LIN {X 0,Y 467.53,Z 286.872,A -85,B 0,C 180,E1 -7582.074,E2 -7582.074} C_VEL
LIN {X 0,Y 467.591,Z 286.865,A -85,B 0,C 180,E1 -7584.888,E2 -7584.888} C_VEL
LIN {X 0,Y 467.615,Z 286.865,A -85,B 0,C 180,E1 -7587.769,E2 -7587.769} C_VEL
LIN {X 0,Y 467.564,Z 286.872,A -85,B 0,C 180,E1 -7591.045,E2 -7591.045} C_VEL
LIN {X 0,Y 467.584,Z 286.87,A -85,B 0,C 180,E1 -7594.242,E2 -7594.242} C_VEL
LIN {X 0,Y 467.545,Z 286.875,A -85,B 0,C 180,E1 -7597.186,E2 -7597.186} C_VEL
LIN {X 0,Y 467.569,Z 286.869,A -85,B 0,C 180,E1 -7600.265,E2 -7600.265} C_VEL
LIN {X 0,Y 467.548,Z 286.875,A -85,B 0,C 180,E1 -7603.745,E2 -7603.745} C_VEL
LIN {X 0,Y 467.586,Z 286.882,A -85,B 0,C 180,E1 -7605.055,E2 -7605.055} C_VEL
LIN {X 0,Y 468.088,Z 290.387,A -85,B 0,C 180,E1 -7607.496,E2 -7607.496} C_VEL
LIN {X 0,Y 468.175,Z 293.918,A -85,B 0,C 180,E1 -7609.798,E2 -7609.798} C_VEL
LIN {X 0,Y 467.977,Z 298.652,A -85,B 0,C 180,E1 -7612.744,E2 -7612.744} C_VEL
LIN {X 0,Y 467.777,Z 303.629,A -85,B 0,C 180,E1 -7615.724,E2 -7615.724} C_VEL
LIN {X 0,Y 467.533,Z 309.782,A -85,B 0,C 180,E1 -7619.264,E2 -7619.264} C_VEL
LIN {X 0,Y 467.277,Z 315.091,A -85,B 0,C 180,E1 -7622.209,E2 -7622.209} C_VEL
LIN {X 0,Y 467.138,Z 320.41,A -85,B 0,C 180,E1 -7625.086,E2 -7625.086} C_VEL
LIN {X 0,Y 466.974,Z 326.319,A -85,B 0,C 180,E1 -7628.206,E2 -7628.206} C_VEL
LIN {X 0,Y 471.454,Z 343.046,A -85,B 0,C 180,E1 -7628.788,E2 -7628.788} C_VEL
LIN {X 0,Y 473.649,Z 353.438,A -85,B 0,C 180,E1 -7629.228,E2 -7629.228} C_VEL
LIN {X 0,Y 473.146,Z 366.892,A -85,B 0,C 180,E1 -7629.767,E2 -7629.767} C_VEL
LIN {X 0,Y 472.348,Z 380.121,A -85,B 0,C 180,E1 -7630.441,E2 -7630.441} C_VEL
LIN {X 0,Y 471.548,Z 393.604,A -85,B 0,C 180,E1 -7631.311,E2 -7631.311} C_VEL
LIN {X 0,Y 470.665,Z 407.326,A -85,B 0,C 180,E1 -7632.4,E2 -7632.4} C_VEL
LIN {X 0,Y 469.85,Z 419.744,A -85,B 0,C 180,E1 -7633.601,E2 -7633.601} C_VEL
LIN {X 0,Y 469.066,Z 430.152,A -85,B 0,C 180,E1 -7634.799,E2 -7634.799} C_VEL
LIN {X 0,Y 468.451,Z 439.813,A -85,B 0,C 180,E1 -7636.111,E2 -7636.111} C_VEL
LIN {X 0,Y 467.819,Z 448.806,A -85,B 0,C 180,E1 -7637.55,E2 -7637.55} C_VEL
LIN {X 0,Y 467.464,Z 457.202,A -85,B 0,C 180,E1 -7639.168,E2 -7639.168} C_VEL
LIN {X 0,Y 467.052,Z 464.577,A -85,B 0,C 180,E1 -7640.909,E2 -7640.909} C_VEL
LIN {X 0,Y 466.824,Z 470.426,A -85,B 0,C 180,E1 -7642.648,E2 -7642.648} C_VEL
LIN {X 0,Y 466.726,Z 473.902,A -85,B 0,C 180,E1 -7643.949,E2 -7643.949} C_VEL
LIN {X 0,Y 466.617,Z 477.414,A -85,B 0,C 180,E1 -7645.681,E2 -7645.681} C_VEL
LIN {X 0,Y 466.638,Z 479.725,A -85,B 0,C 180,E1 -7647.41,E2 -7647.41} C_VEL
LIN {X 0,Y 466.586,Z 480.888,A -85,B 0,C 180,E1 -7649.137,E2 -7649.137} C_VEL
LIN {X 0,Y 466.586,Z 480.887,A -85,B 0,C 180,E1 -7650.863,E2 -7650.863} C_VEL
LIN {X 0,Y 466.638,Z 479.722,A -85,B 0,C 180,E1 -7652.589,E2 -7652.589} C_VEL
LIN {X 0,Y 466.617,Z 477.411,A -85,B 0,C 180,E1 -7654.319,E2 -7654.319} C_VEL
LIN {X 0,Y 466.751,Z 473.905,A -85,B 0,C 180,E1 -7656.05,E2 -7656.05} C_VEL
LIN {X 0,Y 466.862,Z 469.113,A -85,B 0,C 180,E1 -7657.786,E2 -7657.786} C_VEL
LIN {X 0,Y 467.115,Z 462.905,A -85,B 0,C 180,E1 -7659.526,E2 -7659.526} C_VEL
LIN {X 0,Y 467.59,Z 455.107,A -85,B 0,C 180,E1 -7661.267,E2 -7661.267} C_VEL
LIN {X 0,Y 467.983,Z 446.593,A -85,B 0,C 180,E1 -7662.833,E2 -7662.833} C_VEL
LIN {X 0,Y 468.659,Z 436.814,A -85,B 0,C 180,E1 -7664.325,E2 -7664.325} C_VEL
LIN {X 0,Y 469.317,Z 426.585,A -85,B 0,C 180,E1 -7665.637,E2 -7665.637} C_VEL
LIN {X 0,Y 470.163,Z 414.572,A -85,B 0,C 180,E1 -7666.928,E2 -7666.928} C_VEL
LIN {X 0,Y 470.985,Z 402.163,A -85,B 0,C 180,E1 -7668.036,E2 -7668.036} C_VEL
LIN {X 0,Y 471.84,Z 388.848,A -85,B 0,C 180,E1 -7669.015,E2 -7669.015} C_VEL
LIN {X 0,Y 472.717,Z 374.15,A -85,B 0,C 180,E1 -7669.882,E2 -7669.882} C_VEL
LIN {X 0,Y 473.379,Z 360.05,A -85,B 0,C 180,E1 -7670.527,E2 -7670.527} C_VEL
LIN {X 0,Y 473.507,Z 352.11,A -85,B 0,C 180,E1 -7670.827,E2 -7670.827} C_VEL
LIN {X 0,Y 469.977,Z 337.263,A -85,B 0,C 180,E1 -7671.427,E2 -7671.427} C_VEL
LIN {X 0,Y 466.957,Z 326.298,A -85,B 0,C 180,E1 -7671.815,E2 -7671.815} C_VEL
LIN {X 0,Y 467.136,Z 320.455,A -85,B 0,C 180,E1 -7674.913,E2 -7674.913} C_VEL
LIN {X 0,Y 467.277,Z 315.165,A -85,B 0,C 180,E1 -7677.79,E2 -7677.79} C_VEL
LIN {X 0,Y 467.536,Z 309.843,A -85,B 0,C 180,E1 -7680.735,E2 -7680.735} C_VEL
LIN {X 0,Y 467.774,Z 303.655,A -85,B 0,C 180,E1 -7684.276,E2 -7684.276} C_VEL
LIN {X 0,Y 467.974,Z 298.65,A -85,B 0,C 180,E1 -7687.255,E2 -7687.255} C_VEL
LIN {X 0,Y 468.172,Z 293.896,A -85,B 0,C 180,E1 -7690.202,E2 -7690.202} C_VEL
LIN {X 0,Y 468.082,Z 290.182,A -85,B 0,C 180,E1 -7692.633,E2 -7692.633} C_VEL
LIN {X 0,Y 467.585,Z 286.869,A -85,B 0,C 180,E1 -7695.055,E2 -7695.055} C_VEL
LIN {X 0,Y 467.583,Z 286.87,A -85,B 0,C 180,E1 -7697.439,E2 -7697.439} C_VEL
LIN {X 0,Y 467.576,Z 286.867,A -85,B 0,C 180,E1 -7700.855,E2 -7700.855} C_VEL
LIN {X 0,Y 467.552,Z 286.872,A -85,B 0,C 180,E1 -7704.261,E2 -7704.261} C_VEL
LIN {X 0,Y 467.575,Z 286.87,A -85,B 0,C 180,E1 -7707.32,E2 -7707.32} C_VEL
LIN {X 0,Y 467.561,Z 286.873,A -85,B 0,C 180,E1 -7710.667,E2 -7710.667} C_VEL
LIN {X 0,Y 467.608,Z 286.863,A -85,B 0,C 180,E1 -7713.199,E2 -7713.199} C_VEL
LIN {X 0,Y 467.585,Z 286.865,A -85,B 0,C 180,E1 -7716.468,E2 -7716.468} C_VEL
LIN {X 0,Y 467.614,Z 286.863,A -85,B 0,C 180,E1 -7719.777,E2 -7719.777} C_VEL
LIN {X 0,Y 467.6,Z 286.862,A -85,B 0,C 180,E1 -7722.507,E2 -7722.507} C_VEL
LIN {X 0,Y 467.595,Z 286.863,A -85,B 0,C 180,E1 -7725.196,E2 -7725.196} C_VEL
LIN {X 0,Y 467.648,Z 286.859,A -85,B 0,C 180,E1 -7727.854,E2 -7727.854} C_VEL
LIN {X 0,Y 467.663,Z 286.854,A -85,B 0,C 180,E1 -7731.357,E2 -7731.357} C_VEL
LIN {X 0,Y 467.711,Z 286.851,A -85,B 0,C 180,E1 -7733.962,E2 -7733.962} C_VEL
LIN {X 0,Y 467.853,Z 286.829,A -85,B 0,C 180,E1 -7737.417,E2 -7737.417} C_VEL
LIN {X 0,Y 467.871,Z 286.833,A -85,B 0,C 180,E1 -7740,E2 -7740} C_VEL
LIN {X 0,Y 467.853,Z 286.832,A -85,B 0,C 180,E1 -7742.583,E2 -7742.583} C_VEL
LIN {X 0,Y 467.711,Z 286.853,A -85,B 0,C 180,E1 -7746.038,E2 -7746.038} C_VEL
LIN {X 0,Y 467.657,Z 286.858,A -85,B 0,C 180,E1 -7749.515,E2 -7749.515} C_VEL
LIN {X 0,Y 467.645,Z 286.861,A -85,B 0,C 180,E1 -7752.358,E2 -7752.358} C_VEL
LIN {X 0,Y 467.641,Z 286.858,A -85,B 0,C 180,E1 -7755.886,E2 -7755.886} C_VEL
LIN {X 0,Y 467.615,Z 286.861,A -85,B 0,C 180,E1 -7759.308,E2 -7759.308} C_VEL
LIN {X 0,Y 467.527,Z 286.872,A -85,B 0,C 180,E1 -7762.074,E2 -7762.074} C_VEL
LIN {X 0,Y 467.596,Z 286.864,A -85,B 0,C 180,E1 -7764.888,E2 -7764.888} C_VEL
LIN {X 0,Y 467.612,Z 286.862,A -85,B 0,C 180,E1 -7767.77,E2 -7767.77} C_VEL
LIN {X 0,Y 467.562,Z 286.866,A -85,B 0,C 180,E1 -7771.046,E2 -7771.046} C_VEL
LIN {X 0,Y 467.581,Z 286.864,A -85,B 0,C 180,E1 -7774.243,E2 -7774.243} C_VEL
LIN {X 0,Y 467.541,Z 286.871,A -85,B 0,C 180,E1 -7777.187,E2 -7777.187} C_VEL
LIN {X 0,Y 467.572,Z 286.868,A -85,B 0,C 180,E1 -7780.265,E2 -7780.265} C_VEL
LIN {X 0,Y 467.581,Z 286.869,A -85,B 0,C 180,E1 -7782.568,E2 -7782.568} C_VEL
LIN {X 0,Y 467.565,Z 286.868,A -85,B 0,C 180,E1 -7785.054,E2 -7785.054} C_VEL
LIN {X 0,Y 467.548,Z 286.873,A -85,B 0,C 180,E1 -7786.256,E2 -7786.256} C_VEL
LIN {X 0,Y 467.686,Z 287.984,A -85,B 0,C 180,E1 -7787.452,E2 -7787.452} C_VEL
LIN {X 0,Y 467.824,Z 291.312,A -85,B 0,C 180,E1 -7790.011,E2 -7790.011} C_VEL
LIN {X 0,Y 467.65,Z 295.467,A -85,B 0,C 180,E1 -7793.05,E2 -7793.05} C_VEL
LIN {X 0,Y 467.496,Z 299.944,A -85,B 0,C 180,E1 -7796.205,E2 -7796.205} C_VEL
LIN {X 0,Y 467.362,Z 304.407,A -85,B 0,C 180,E1 -7799.252,E2 -7799.252} C_VEL
LIN {X 0,Y 467.18,Z 309.443,A -85,B 0,C 180,E1 -7802.569,E2 -7802.569} C_VEL
LIN {X 0,Y 467.068,Z 313.378,A -85,B 0,C 180,E1 -7805.083,E2 -7805.083} C_VEL
LIN {X 0,Y 466.904,Z 318.442,A -85,B 0,C 180,E1 -7808.249,E2 -7808.249} C_VEL
LIN {X 0,Y 471.953,Z 336.104,A -85,B 0,C 180,E1 -7808.906,E2 -7808.906} C_VEL
LIN {X 0,Y 473.76,Z 344.418,A -85,B 0,C 180,E1 -7809.263,E2 -7809.263} C_VEL
LIN {X 0,Y 473.225,Z 358.757,A -85,B 0,C 180,E1 -7809.841,E2 -7809.841} C_VEL
LIN {X 0,Y 472.462,Z 371.728,A -85,B 0,C 180,E1 -7810.51,E2 -7810.51} C_VEL
LIN {X 0,Y 471.49,Z 377.067,A -85,B 0,C 180,E1 -7810.802,E2 -7810.802} C_VEL
LIN {X 0,Y 468.181,Z 385.652,A -85,B 0,C 180,E1 -7811.268,E2 -7811.268} C_VEL
LIN {X 0,Y 464.911,Z 393.932,A -85,B 0,C 180,E1 -7811.8,E2 -7811.8} C_VEL
LIN {X 0,Y 463.993,Z 398.749,A -85,B 0,C 180,E1 -7812.191,E2 -7812.191} C_VEL
LIN {X 0,Y 463.059,Z 411.677,A -85,B 0,C 180,E1 -7813.467,E2 -7813.467} C_VEL
LIN {X 0,Y 462.213,Z 422.838,A -85,B 0,C 180,E1 -7814.795,E2 -7814.795} C_VEL
LIN {X 0,Y 461.403,Z 433.683,A -85,B 0,C 180,E1 -7816.345,E2 -7816.345} C_VEL
LIN {X 0,Y 460.798,Z 442.684,A -85,B 0,C 180,E1 -7817.895,E2 -7817.895} C_VEL
LIN {X 0,Y 460.326,Z 450.145,A -85,B 0,C 180,E1 -7819.444,E2 -7819.444} C_VEL
LIN {X 0,Y 460.001,Z 457.122,A -85,B 0,C 180,E1 -7821.212,E2 -7821.212} C_VEL
LIN {X 0,Y 459.74,Z 462.608,A -85,B 0,C 180,E1 -7822.976,E2 -7822.976} C_VEL
LIN {X 0,Y 459.643,Z 466.751,A -85,B 0,C 180,E1 -7824.737,E2 -7824.737} C_VEL
LIN {X 0,Y 459.57,Z 469.665,A -85,B 0,C 180,E1 -7826.493,E2 -7826.493} C_VEL
LIN {X 0,Y 459.518,Z 471.42,A -85,B 0,C 180,E1 -7828.247,E2 -7828.247} C_VEL
LIN {X 0,Y 459.499,Z 472.035,A -85,B 0,C 180,E1 -7830,E2 -7830} C_VEL
LIN {X 0,Y 459.518,Z 471.472,A -85,B 0,C 180,E1 -7831.753,E2 -7831.753} C_VEL
LIN {X 0,Y 459.571,Z 469.785,A -85,B 0,C 180,E1 -7833.507,E2 -7833.507} C_VEL
LIN {X 0,Y 459.635,Z 466.935,A -85,B 0,C 180,E1 -7835.264,E2 -7835.264} C_VEL
LIN {X 0,Y 459.735,Z 462.856,A -85,B 0,C 180,E1 -7837.025,E2 -7837.025} C_VEL
LIN {X 0,Y 459.976,Z 457.447,A -85,B 0,C 180,E1 -7838.789,E2 -7838.789} C_VEL
LIN {X 0,Y 460.314,Z 450.557,A -85,B 0,C 180,E1 -7840.557,E2 -7840.557} C_VEL
LIN {X 0,Y 460.769,Z 443.148,A -85,B 0,C 180,E1 -7842.106,E2 -7842.106} C_VEL
LIN {X 0,Y 461.341,Z 434.225,A -85,B 0,C 180,E1 -7843.658,E2 -7843.658} C_VEL
LIN {X 0,Y 462.021,Z 425.129,A -85,B 0,C 180,E1 -7844.987,E2 -7844.987} C_VEL
LIN {X 0,Y 462.838,Z 414.4,A -85,B 0,C 180,E1 -7846.315,E2 -7846.315} C_VEL
LIN {X 0,Y 463.683,Z 403.336,A -85,B 0,C 180,E1 -7847.47,E2 -7847.47} C_VEL
LIN {X 0,Y 464.521,Z 391.329,A -85,B 0,C 180,E1 -7848.525,E2 -7848.525} C_VEL
LIN {X 0,Y 465.39,Z 377.565,A -85,B 0,C 180,E1 -7849.519,E2 -7849.519} C_VEL
LIN {X 0,Y 466.313,Z 363.297,A -85,B 0,C 180,E1 -7850.335,E2 -7850.335} C_VEL
LIN {X 0,Y 466.865,Z 350.144,A -85,B 0,C 180,E1 -7850.932,E2 -7850.932} C_VEL
LIN {X 0,Y 466.952,Z 344.718,A -85,B 0,C 180,E1 -7851.136,E2 -7851.136} C_VEL
LIN {X 0,Y 463.432,Z 330.804,A -85,B 0,C 180,E1 -7851.741,E2 -7851.741} C_VEL
LIN {X 0,Y 459.865,Z 318.523,A -85,B 0,C 180,E1 -7852.202,E2 -7852.202} C_VEL
LIN {X 0,Y 460.037,Z 313.638,A -85,B 0,C 180,E1 -7855.325,E2 -7855.325} C_VEL
LIN {X 0,Y 460.153,Z 309.162,A -85,B 0,C 180,E1 -7858.26,E2 -7858.26} C_VEL
LIN {X 0,Y 460.333,Z 304.672,A -85,B 0,C 180,E1 -7861.271,E2 -7861.271} C_VEL
LIN {X 0,Y 460.537,Z 299.988,A -85,B 0,C 180,E1 -7864.506,E2 -7864.506} C_VEL
LIN {X 0,Y 460.635,Z 295.664,A -85,B 0,C 180,E1 -7867.61,E2 -7867.61} C_VEL
LIN {X 0,Y 460.812,Z 292.023,A -85,B 0,C 180,E1 -7870.309,E2 -7870.309} C_VEL
LIN {X 0,Y 460.627,Z 288.705,A -85,B 0,C 180,E1 -7872.915,E2 -7872.915} C_VEL
LIN {X 0,Y 460.535,Z 288.146,A -85,B 0,C 180,E1 -7873.371,E2 -7873.371} C_VEL
LIN {X 0,Y 460.516,Z 287.75,A -85,B 0,C 180,E1 -7874.588,E2 -7874.588} C_VEL
LIN {X 0,Y 460.522,Z 287.746,A -85,B 0,C 180,E1 -7877.818,E2 -7877.818} C_VEL
LIN {X 0,Y 460.543,Z 287.743,A -85,B 0,C 180,E1 -7881.102,E2 -7881.102} C_VEL
LIN {X 0,Y 460.507,Z 287.75,A -85,B 0,C 180,E1 -7884.554,E2 -7884.554} C_VEL
LIN {X 0,Y 460.528,Z 287.748,A -85,B 0,C 180,E1 -7887.715,E2 -7887.715} C_VEL
LIN {X 0,Y 460.524,Z 287.747,A -85,B 0,C 180,E1 -7890.768,E2 -7890.768} C_VEL
LIN {X 0,Y 460.528,Z 287.744,A -85,B 0,C 180,E1 -7893.732,E2 -7893.732} C_VEL
LIN {X 0,Y 460.541,Z 287.743,A -85,B 0,C 180,E1 -7896.624,E2 -7896.624} C_VEL
LIN {X 0,Y 460.548,Z 287.742,A -85,B 0,C 180,E1 -7899.452,E2 -7899.452} C_VEL
LIN {X 0,Y 460.556,Z 287.741,A -85,B 0,C 180,E1 -7902.23,E2 -7902.23} C_VEL
LIN {X 0,Y 460.559,Z 287.743,A -85,B 0,C 180,E1 -7904.965,E2 -7904.965} C_VEL
LIN {X 0,Y 460.608,Z 287.734,A -85,B 0,C 180,E1 -7908.559,E2 -7908.559} C_VEL
LIN {X 0,Y 460.618,Z 287.733,A -85,B 0,C 180,E1 -7911.224,E2 -7911.224} C_VEL
LIN {X 0,Y 460.679,Z 287.728,A -85,B 0,C 180,E1 -7913.87,E2 -7913.87} C_VEL
LIN {X 0,Y 460.822,Z 287.708,A -85,B 0,C 180,E1 -7917.378,E2 -7917.378} C_VEL
LIN {X 0,Y 460.845,Z 287.708,A -85,B 0,C 180,E1 -7920,E2 -7920} C_VEL
LIN {X 0,Y 460.822,Z 287.708,A -85,B 0,C 180,E1 -7922.622,E2 -7922.622} C_VEL
LIN {X 0,Y 460.679,Z 287.729,A -85,B 0,C 180,E1 -7926.13,E2 -7926.13} C_VEL
LIN {X 0,Y 460.618,Z 287.733,A -85,B 0,C 180,E1 -7928.776,E2 -7928.776} C_VEL
LIN {X 0,Y 460.61,Z 287.737,A -85,B 0,C 180,E1 -7932.445,E2 -7932.445} C_VEL
LIN {X 0,Y 460.597,Z 287.735,A -85,B 0,C 180,E1 -7935.998,E2 -7935.998} C_VEL
LIN {X 0,Y 460.567,Z 287.739,A -85,B 0,C 180,E1 -7938.902,E2 -7938.902} C_VEL
LIN {X 0,Y 460.512,Z 287.75,A -85,B 0,C 180,E1 -7941.486,E2 -7941.486} C_VEL
LIN {X 0,Y 460.535,Z 287.746,A -85,B 0,C 180,E1 -7944.333,E2 -7944.333} C_VEL
LIN {X 0,Y 460.568,Z 287.741,A -85,B 0,C 180,E1 -7947.244,E2 -7947.244} C_VEL
LIN {X 0,Y 460.506,Z 287.751,A -85,B 0,C 180,E1 -7950.24,E2 -7950.24} C_VEL
LIN {X 0,Y 460.524,Z 287.75,A -85,B 0,C 180,E1 -7953.325,E2 -7953.325} C_VEL
LIN {X 0,Y 460.473,Z 287.758,A -85,B 0,C 180,E1 -7956.53,E2 -7956.53} C_VEL
LIN {X 0,Y 460.52,Z 287.751,A -85,B 0,C 180,E1 -7959.863,E2 -7959.863} C_VEL
LIN {X 0,Y 460.49,Z 287.753,A -85,B 0,C 180,E1 -7962.898,E2 -7962.898} C_VEL
LIN {X 0,Y 460.581,Z 287.869,A -85,B 0,C 180,E1 -7964.903,E2 -7964.903} C_VEL
LIN {X 0,Y 461.025,Z 290.861,A -85,B 0,C 180,E1 -7967.031,E2 -7967.031} C_VEL
LIN {X 0,Y 461.154,Z 294.773,A -85,B 0,C 180,E1 -7969.641,E2 -7969.641} C_VEL
LIN {X 0,Y 460.966,Z 299.196,A -85,B 0,C 180,E1 -7972.448,E2 -7972.448} C_VEL
LIN {X 0,Y 460.755,Z 304.442,A -85,B 0,C 180,E1 -7975.642,E2 -7975.642} C_VEL
LIN {X 0,Y 460.502,Z 309.727,A -85,B 0,C 180,E1 -7978.742,E2 -7978.742} C_VEL
LIN {X 0,Y 460.252,Z 315.041,A -85,B 0,C 180,E1 -7981.747,E2 -7981.747} C_VEL
LIN {X 0,Y 460.109,Z 320.346,A -85,B 0,C 180,E1 -7984.679,E2 -7984.679} C_VEL
LIN {X 0,Y 459.921,Z 326.247,A -85,B 0,C 180,E1 -7987.851,E2 -7987.851} C_VEL
LIN {X 0,Y 464.622,Z 343.544,A -85,B 0,C 180,E1 -7988.477,E2 -7988.477} C_VEL
LIN {X 0,Y 466.935,Z 354.818,A -85,B 0,C 180,E1 -7988.97,E2 -7988.97} C_VEL
LIN {X 0,Y 466.413,Z 368.196,A -85,B 0,C 180,E1 -7989.531,E2 -7989.531} C_VEL
LIN {X 0,Y 465.518,Z 381.867,A -85,B 0,C 180,E1 -7990.257,E2 -7990.257} C_VEL
LIN {X 0,Y 464.699,Z 395.053,A -85,B 0,C 180,E1 -7991.139,E2 -7991.139} C_VEL
LIN {X 0,Y 463.774,Z 408.475,A -85,B 0,C 180,E1 -7992.243,E2 -7992.243} C_VEL
LIN {X 0,Y 462.917,Z 420.695,A -85,B 0,C 180,E1 -7993.461,E2 -7993.461} C_VEL
LIN {X 0,Y 462.054,Z 431.85,A -85,B 0,C 180,E1 -7994.789,E2 -7994.789} C_VEL
LIN {X 0,Y 461.277,Z 442.671,A -85,B 0,C 180,E1 -7996.34,E2 -7996.34} C_VEL
LIN {X 0,Y 460.663,Z 451.681,A -85,B 0,C 180,E1 -7997.891,E2 -7997.891} C_VEL
LIN {X 0,Y 460.275,Z 459.153,A -85,B 0,C 180,E1 -7999.442,E2 -7999.442} C_VEL
LIN {X 0,Y 459.918,Z 466.123,A -85,B 0,C 180,E1 -8001.21,E2 -8001.21} C_VEL
LIN {X 0,Y 459.73,Z 471.602,A -85,B 0,C 180,E1 -8002.975,E2 -8002.975} C_VEL
LIN {X 0,Y 459.606,Z 475.744,A -85,B 0,C 180,E1 -8004.736,E2 -8004.736} C_VEL
LIN {X 0,Y 459.538,Z 478.647,A -85,B 0,C 180,E1 -8006.492,E2 -8006.492} C_VEL
LIN {X 0,Y 459.513,Z 480.379,A -85,B 0,C 180,E1 -8008.247,E2 -8008.247} C_VEL
LIN {X 0,Y 459.498,Z 480.972,A -85,B 0,C 180,E1 -8010,E2 -8010} C_VEL
LIN {X 0,Y 459.513,Z 480.377,A -85,B 0,C 180,E1 -8011.753,E2 -8011.753} C_VEL
LIN {X 0,Y 459.537,Z 478.642,A -85,B 0,C 180,E1 -8013.507,E2 -8013.507} C_VEL
LIN {X 0,Y 459.612,Z 475.743,A -85,B 0,C 180,E1 -8015.264,E2 -8015.264} C_VEL
LIN {X 0,Y 459.734,Z 471.607,A -85,B 0,C 180,E1 -8017.024,E2 -8017.024} C_VEL
LIN {X 0,Y 459.917,Z 466.125,A -85,B 0,C 180,E1 -8018.789,E2 -8018.789} C_VEL
LIN {X 0,Y 460.274,Z 459.148,A -85,B 0,C 180,E1 -8020.557,E2 -8020.557} C_VEL
LIN {X 0,Y 460.687,Z 451.678,A -85,B 0,C 180,E1 -8022.108,E2 -8022.108} C_VEL
LIN {X 0,Y 461.275,Z 442.672,A -85,B 0,C 180,E1 -8023.659,E2 -8023.659} C_VEL
LIN {X 0,Y 462.029,Z 431.848,A -85,B 0,C 180,E1 -8025.211,E2 -8025.211} C_VEL
LIN {X 0,Y 462.962,Z 419.679,A -85,B 0,C 180,E1 -8026.65,E2 -8026.65} C_VEL
LIN {X 0,Y 463.864,Z 407.265,A -85,B 0,C 180,E1 -8027.866,E2 -8027.866} C_VEL
LIN {X 0,Y 464.781,Z 393.528,A -85,B 0,C 180,E1 -8028.971,E2 -8028.971} C_VEL
LIN {X 0,Y 465.675,Z 380.037,A -85,B 0,C 180,E1 -8029.85,E2 -8029.85} C_VEL
LIN {X 0,Y 466.494,Z 365.036,A -85,B 0,C 180,E1 -8030.62,E2 -8030.62} C_VEL
LIN {X 0,Y 466.853,Z 353.513,A -85,B 0,C 180,E1 -8031.082,E2 -8031.082} C_VEL
LIN {X 0,Y 463.334,Z 338.697,A -85,B 0,C 180,E1 -8031.711,E2 -8031.711} C_VEL
LIN {X 0,Y 459.903,Z 326.243,A -85,B 0,C 180,E1 -8032.159,E2 -8032.159} C_VEL
LIN {X 0,Y 460.107,Z 320.394,A -85,B 0,C 180,E1 -8035.32,E2 -8035.32} C_VEL
LIN {X 0,Y 460.251,Z 315.106,A -85,B 0,C 180,E1 -8038.252,E2 -8038.252} C_VEL
LIN {X 0,Y 460.491,Z 309.758,A -85,B 0,C 180,E1 -8041.277,E2 -8041.277} C_VEL
LIN {X 0,Y 460.741,Z 304.156,A -85,B 0,C 180,E1 -8044.543,E2 -8044.543} C_VEL
LIN {X 0,Y 460.964,Z 299.155,A -85,B 0,C 180,E1 -8047.578,E2 -8047.578} C_VEL
LIN {X 0,Y 461.15,Z 294.758,A -85,B 0,C 180,E1 -8050.359,E2 -8050.359} C_VEL
LIN {X 0,Y 461.018,Z 290.857,A -85,B 0,C 180,E1 -8052.968,E2 -8052.968} C_VEL
LIN {X 0,Y 460.536,Z 287.747,A -85,B 0,C 180,E1 -8055.198,E2 -8055.198} C_VEL
LIN {X 0,Y 460.526,Z 287.749,A -85,B 0,C 180,E1 -8058.397,E2 -8058.397} C_VEL
LIN {X 0,Y 460.52,Z 287.747,A -85,B 0,C 180,E1 -8061.266,E2 -8061.266} C_VEL
LIN {X 0,Y 460.502,Z 287.752,A -85,B 0,C 180,E1 -8064.554,E2 -8064.554} C_VEL
LIN {X 0,Y 460.525,Z 287.751,A -85,B 0,C 180,E1 -8067.715,E2 -8067.715} C_VEL
LIN {X 0,Y 460.531,Z 287.75,A -85,B 0,C 180,E1 -8070.769,E2 -8070.769} C_VEL
LIN {X 0,Y 460.555,Z 287.744,A -85,B 0,C 180,E1 -8073.734,E2 -8073.734} C_VEL
LIN {X 0,Y 460.538,Z 287.743,A -85,B 0,C 180,E1 -8076.624,E2 -8076.624} C_VEL
LIN {X 0,Y 460.543,Z 287.742,A -85,B 0,C 180,E1 -8079.452,E2 -8079.452} C_VEL
LIN {X 0,Y 460.55,Z 287.74,A -85,B 0,C 180,E1 -8082.23,E2 -8082.23} C_VEL
LIN {X 0,Y 460.555,Z 287.741,A -85,B 0,C 180,E1 -8084.965,E2 -8084.965} C_VEL
LIN {X 0,Y 460.606,Z 287.733,A -85,B 0,C 180,E1 -8088.559,E2 -8088.559} C_VEL
LIN {X 0,Y 460.614,Z 287.733,A -85,B 0,C 180,E1 -8091.224,E2 -8091.224} C_VEL
LIN {X 0,Y 460.675,Z 287.728,A -85,B 0,C 180,E1 -8093.87,E2 -8093.87} C_VEL
LIN {X 0,Y 460.818,Z 287.706,A -85,B 0,C 180,E1 -8097.378,E2 -8097.378} C_VEL
LIN {X 0,Y 460.842,Z 287.709,A -85,B 0,C 180,E1 -8100,E2 -8100} C_VEL
LIN {X 0,Y 460.818,Z 287.708,A -85,B 0,C 180,E1 -8102.622,E2 -8102.622} C_VEL
LIN {X 0,Y 460.675,Z 287.73,A -85,B 0,C 180,E1 -8106.13,E2 -8106.13} C_VEL
LIN {X 0,Y 460.613,Z 287.732,A -85,B 0,C 180,E1 -8108.777,E2 -8108.777} C_VEL
LIN {X 0,Y 460.605,Z 287.737,A -85,B 0,C 180,E1 -8112.445,E2 -8112.445} C_VEL
LIN {X 0,Y 460.592,Z 287.736,A -85,B 0,C 180,E1 -8115.998,E2 -8115.998} C_VEL
LIN {X 0,Y 460.563,Z 287.74,A -85,B 0,C 180,E1 -8118.902,E2 -8118.902} C_VEL
LIN {X 0,Y 460.508,Z 287.75,A -85,B 0,C 180,E1 -8121.486,E2 -8121.486} C_VEL
LIN {X 0,Y 460.535,Z 287.746,A -85,B 0,C 180,E1 -8124.333,E2 -8124.333} C_VEL
LIN {X 0,Y 460.565,Z 287.74,A -85,B 0,C 180,E1 -8127.244,E2 -8127.244} C_VEL
LIN {X 0,Y 460.504,Z 287.746,A -85,B 0,C 180,E1 -8130.241,E2 -8130.241} C_VEL
LIN {X 0,Y 460.523,Z 287.744,A -85,B 0,C 180,E1 -8133.326,E2 -8133.326} C_VEL
LIN {X 0,Y 460.47,Z 287.753,A -85,B 0,C 180,E1 -8136.53,E2 -8136.53} C_VEL
LIN {X 0,Y 460.553,Z 287.745,A -85,B 0,C 180,E1 -8139.86,E2 -8139.86} C_VEL
LIN {X 0,Y 460.508,Z 287.751,A -85,B 0,C 180,E1 -8142.901,E2 -8142.901} C_VEL
LIN {X 0,Y 460.504,Z 287.751,A -85,B 0,C 180,E1 -8145.831,E2 -8145.831} C_VEL
LIN {X 0,Y 460.514,Z 288.014,A -85,B 0,C 180,E1 -8146.628,E2 -8146.628} C_VEL
LIN {X 0,Y 460.779,Z 291.025,A -85,B 0,C 180,E1 -8149.017,E2 -8149.017} C_VEL
LIN {X 0,Y 460.678,Z 294.016,A -85,B 0,C 180,E1 -8151.283,E2 -8151.283} C_VEL
LIN {X 0,Y 460.537,Z 298.499,A -85,B 0,C 180,E1 -8154.558,E2 -8154.558} C_VEL
LIN {X 0,Y 460.335,Z 302.974,A -85,B 0,C 180,E1 -8157.701,E2 -8157.701} C_VEL
LIN {X 0,Y 460.234,Z 307.436,A -85,B 0,C 180,E1 -8160.749,E2 -8160.749} C_VEL
LIN {X 0,Y 460.042,Z 311.939,A -85,B 0,C 180,E1 -8163.704,E2 -8163.704} C_VEL
LIN {X 0,Y 459.927,Z 316.443,A -85,B 0,C 180,E1 -8166.591,E2 -8166.591} C_VEL
LIN {X 0,Y 459.889,Z 318.687,A -85,B 0,C 180,E1 -8167.915,E2 -8167.915} C_VEL
LIN {X 0,Y 464.613,Z 334.925,A -85,B 0,C 180,E1 -8168.516,E2 -8168.516} C_VEL
LIN {X 0,Y 467.085,Z 345.773,A -85,B 0,C 180,E1 -8169.001,E2 -8169.001} C_VEL
LIN {X 0,Y 466.449,Z 360.857,A -85,B 0,C 180,E1 -8169.638,E2 -8169.638} C_VEL
LIN {X 0,Y 465.594,Z 374.4,A -85,B 0,C 180,E1 -8170.376,E2 -8170.376} C_VEL
LIN {X 0,Y 464.783,Z 387.356,A -85,B 0,C 180,E1 -8171.258,E2 -8171.258} C_VEL
LIN {X 0,Y 463.993,Z 398.749,A -85,B 0,C 180,E1 -8172.191,E2 -8172.191} C_VEL
LIN {X 0,Y 463.063,Z 403.536,A -85,B 0,C 180,E1 -8172.608,E2 -8172.608} C_VEL
LIN {X 0,Y 459.705,Z 411.168,A -85,B 0,C 180,E1 -8173.283,E2 -8173.283} C_VEL
LIN {X 0,Y 456.325,Z 418.431,A -85,B 0,C 180,E1 -8174.016,E2 -8174.016} C_VEL
LIN {X 0,Y 455.358,Z 422.589,A -85,B 0,C 180,E1 -8174.519,E2 -8174.519} C_VEL
LIN {X 0,Y 454.447,Z 433.756,A -85,B 0,C 180,E1 -8176.131,E2 -8176.131} C_VEL
LIN {X 0,Y 453.789,Z 442.756,A -85,B 0,C 180,E1 -8177.705,E2 -8177.705} C_VEL
LIN {X 0,Y 453.324,Z 450.217,A -85,B 0,C 180,E1 -8179.279,E2 -8179.279} C_VEL
LIN {X 0,Y 452.94,Z 457.194,A -85,B 0,C 180,E1 -8181.074,E2 -8181.074} C_VEL
LIN {X 0,Y 452.666,Z 462.679,A -85,B 0,C 180,E1 -8182.866,E2 -8182.866} C_VEL
LIN {X 0,Y 452.56,Z 466.822,A -85,B 0,C 180,E1 -8184.654,E2 -8184.654} C_VEL
LIN {X 0,Y 452.468,Z 469.735,A -85,B 0,C 180,E1 -8186.438,E2 -8186.438} C_VEL
LIN {X 0,Y 452.434,Z 471.49,A -85,B 0,C 180,E1 -8188.22,E2 -8188.22} C_VEL
LIN {X 0,Y 452.405,Z 472.104,A -85,B 0,C 180,E1 -8190,E2 -8190} C_VEL
LIN {X 0,Y 452.435,Z 471.54,A -85,B 0,C 180,E1 -8191.781,E2 -8191.781} C_VEL
LIN {X 0,Y 452.468,Z 469.853,A -85,B 0,C 180,E1 -8193.562,E2 -8193.562} C_VEL
LIN {X 0,Y 452.549,Z 467.003,A -85,B 0,C 180,E1 -8195.347,E2 -8195.347} C_VEL
LIN {X 0,Y 452.662,Z 462.924,A -85,B 0,C 180,E1 -8197.135,E2 -8197.135} C_VEL
LIN {X 0,Y 452.92,Z 457.515,A -85,B 0,C 180,E1 -8198.927,E2 -8198.927} C_VEL
LIN {X 0,Y 453.314,Z 450.624,A -85,B 0,C 180,E1 -8200.722,E2 -8200.722} C_VEL
LIN {X 0,Y 453.759,Z 443.215,A -85,B 0,C 180,E1 -8202.296,E2 -8202.296} C_VEL
LIN {X 0,Y 454.397,Z 434.291,A -85,B 0,C 180,E1 -8203.871,E2 -8203.871} C_VEL
LIN {X 0,Y 455.137,Z 425.194,A -85,B 0,C 180,E1 -8205.219,E2 -8205.219} C_VEL
LIN {X 0,Y 456.004,Z 414.465,A -85,B 0,C 180,E1 -8206.566,E2 -8206.566} C_VEL
LIN {X 0,Y 456.934,Z 402.67,A -85,B 0,C 180,E1 -8207.808,E2 -8207.808} C_VEL
LIN {X 0,Y 457.883,Z 389.97,A -85,B 0,C 180,E1 -8208.92,E2 -8208.92} C_VEL
LIN {X 0,Y 458.681,Z 377.627,A -85,B 0,C 180,E1 -8209.816,E2 -8209.816} C_VEL
LIN {X 0,Y 459.595,Z 364.386,A -85,B 0,C 180,E1 -8210.592,E2 -8210.592} C_VEL
LIN {X 0,Y 460.204,Z 350.682,A -85,B 0,C 180,E1 -8211.228,E2 -8211.228} C_VEL
LIN {X 0,Y 460.239,Z 345.951,A -85,B 0,C 180,E1 -8211.414,E2 -8211.414} C_VEL
LIN {X 0,Y 456.873,Z 332.555,A -85,B 0,C 180,E1 -8212.025,E2 -8212.025} C_VEL
LIN {X 0,Y 452.8,Z 318.583,A -85,B 0,C 180,E1 -8212.57,E2 -8212.57} C_VEL
LIN {X 0,Y 452.961,Z 313.546,A -85,B 0,C 180,E1 -8215.854,E2 -8215.854} C_VEL
LIN {X 0,Y 453.126,Z 309.213,A -85,B 0,C 180,E1 -8218.738,E2 -8218.738} C_VEL
LIN {X 0,Y 453.268,Z 304.73,A -85,B 0,C 180,E1 -8221.815,E2 -8221.815} C_VEL
LIN {X 0,Y 453.504,Z 300.217,A -85,B 0,C 180,E1 -8224.987,E2 -8224.987} C_VEL
LIN {X 0,Y 453.622,Z 295.702,A -85,B 0,C 180,E1 -8228.296,E2 -8228.296} C_VEL
LIN {X 0,Y 453.789,Z 292.615,A -85,B 0,C 180,E1 -8230.634,E2 -8230.634} C_VEL
LIN {X 0,Y 453.539,Z 289.351,A -85,B 0,C 180,E1 -8233.255,E2 -8233.255} C_VEL
LIN {X 0,Y 453.486,Z 288.626,A -85,B 0,C 180,E1 -8234.529,E2 -8234.529} C_VEL
LIN {X 0,Y 453.478,Z 288.624,A -85,B 0,C 180,E1 -8238.209,E2 -8238.209} C_VEL
LIN {X 0,Y 453.514,Z 288.619,A -85,B 0,C 180,E1 -8240.79,E2 -8240.79} C_VEL
LIN {X 0,Y 453.452,Z 288.628,A -85,B 0,C 180,E1 -8243.917,E2 -8243.917} C_VEL
LIN {X 0,Y 453.479,Z 288.623,A -85,B 0,C 180,E1 -8247.151,E2 -8247.151} C_VEL
LIN {X 0,Y 453.464,Z 288.624,A -85,B 0,C 180,E1 -8250.267,E2 -8250.267} C_VEL
LIN {X 0,Y 453.468,Z 288.622,A -85,B 0,C 180,E1 -8253.291,E2 -8253.291} C_VEL
LIN {X 0,Y 453.494,Z 288.62,A -85,B 0,C 180,E1 -8256.238,E2 -8256.238} C_VEL
LIN {X 0,Y 453.479,Z 288.623,A -85,B 0,C 180,E1 -8259.117,E2 -8259.117} C_VEL
LIN {X 0,Y 453.509,Z 288.621,A -85,B 0,C 180,E1 -8261.944,E2 -8261.944} C_VEL
LIN {X 0,Y 453.535,Z 288.617,A -85,B 0,C 180,E1 -8264.726,E2 -8264.726} C_VEL
LIN {X 0,Y 453.557,Z 288.613,A -85,B 0,C 180,E1 -8268.379,E2 -8268.379} C_VEL
LIN {X 0,Y 453.584,Z 288.611,A -85,B 0,C 180,E1 -8271.086,E2 -8271.086} C_VEL
LIN {X 0,Y 453.645,Z 288.604,A -85,B 0,C 180,E1 -8273.774,E2 -8273.774} C_VEL
LIN {X 0,Y 453.762,Z 288.588,A -85,B 0,C 180,E1 -8277.337,E2 -8277.337} C_VEL
LIN {X 0,Y 453.815,Z 288.584,A -85,B 0,C 180,E1 -8280,E2 -8280} C_VEL
LIN {X 0,Y 453.763,Z 288.588,A -85,B 0,C 180,E1 -8282.663,E2 -8282.663} C_VEL
LIN {X 0,Y 453.645,Z 288.605,A -85,B 0,C 180,E1 -8286.226,E2 -8286.226} C_VEL
LIN {X 0,Y 453.584,Z 288.611,A -85,B 0,C 180,E1 -8288.913,E2 -8288.913} C_VEL
LIN {X 0,Y 453.56,Z 288.615,A -85,B 0,C 180,E1 -8292.529,E2 -8292.529} C_VEL
LIN {X 0,Y 453.541,Z 288.614,A -85,B 0,C 180,E1 -8296.196,E2 -8296.196} C_VEL
LIN {X 0,Y 453.516,Z 288.617,A -85,B 0,C 180,E1 -8299.04,E2 -8299.04} C_VEL
LIN {X 0,Y 453.473,Z 288.624,A -85,B 0,C 180,E1 -8301.836,E2 -8301.836} C_VEL
LIN {X 0,Y 453.504,Z 288.621,A -85,B 0,C 180,E1 -8304.735,E2 -8304.735} C_VEL
LIN {X 0,Y 453.528,Z 288.619,A -85,B 0,C 180,E1 -8307.959,E2 -8307.959} C_VEL
LIN {X 0,Y 453.462,Z 288.628,A -85,B 0,C 180,E1 -8311.525,E2 -8311.525} C_VEL
LIN {X 0,Y 453.484,Z 288.628,A -85,B 0,C 180,E1 -8314.777,E2 -8314.777} C_VEL
LIN {X 0,Y 453.457,Z 288.632,A -85,B 0,C 180,E1 -8318.312,E2 -8318.312} C_VEL
LIN {X 0,Y 453.491,Z 288.623,A -85,B 0,C 180,E1 -8320.609,E2 -8320.609} C_VEL
LIN {X 0,Y 453.466,Z 288.632,A -85,B 0,C 180,E1 -8324.221,E2 -8324.221} C_VEL
LIN {X 0,Y 453.514,Z 288.808,A -85,B 0,C 180,E1 -8324.704,E2 -8324.704} C_VEL
LIN {X 0,Y 454.022,Z 292.083,A -85,B 0,C 180,E1 -8327.071,E2 -8327.071} C_VEL
LIN {X 0,Y 454.142,Z 295.602,A -85,B 0,C 180,E1 -8329.461,E2 -8329.461} C_VEL
LIN {X 0,Y 453.95,Z 299.752,A -85,B 0,C 180,E1 -8332.146,E2 -8332.146} C_VEL
LIN {X 0,Y 453.73,Z 304.626,A -85,B 0,C 180,E1 -8335.179,E2 -8335.179} C_VEL
LIN {X 0,Y 453.462,Z 309.676,A -85,B 0,C 180,E1 -8338.201,E2 -8338.201} C_VEL
LIN {X 0,Y 453.242,Z 314.975,A -85,B 0,C 180,E1 -8341.27,E2 -8341.27} C_VEL
LIN {X 0,Y 453.037,Z 320.284,A -85,B 0,C 180,E1 -8344.255,E2 -8344.255} C_VEL
LIN {X 0,Y 452.868,Z 326.173,A -85,B 0,C 180,E1 -8347.485,E2 -8347.485} C_VEL
LIN {X 0,Y 457.568,Z 343.253,A -85,B 0,C 180,E1 -8348.121,E2 -8348.121} C_VEL
LIN {X 0,Y 460.276,Z 355.769,A -85,B 0,C 180,E1 -8348.69,E2 -8348.69} C_VEL
LIN {X 0,Y 459.662,Z 370.188,A -85,B 0,C 180,E1 -8349.323,E2 -8349.323} C_VEL
LIN {X 0,Y 458.723,Z 383.57,A -85,B 0,C 180,E1 -8350.069,E2 -8350.069} C_VEL
LIN {X 0,Y 457.719,Z 397.84,A -85,B 0,C 180,E1 -8351.073,E2 -8351.073} C_VEL
LIN {X 0,Y 456.781,Z 410.681,A -85,B 0,C 180,E1 -8352.186,E2 -8352.186} C_VEL
LIN {X 0,Y 455.892,Z 422.582,A -85,B 0,C 180,E1 -8353.429,E2 -8353.429} C_VEL
LIN {X 0,Y 455.012,Z 433.414,A -85,B 0,C 180,E1 -8354.777,E2 -8354.777} C_VEL
LIN {X 0,Y 454.22,Z 443.959,A -85,B 0,C 180,E1 -8356.352,E2 -8356.352} C_VEL
LIN {X 0,Y 453.581,Z 452.733,A -85,B 0,C 180,E1 -8357.926,E2 -8357.926} C_VEL
LIN {X 0,Y 453.271,Z 459.085,A -85,B 0,C 180,E1 -8359.277,E2 -8359.277} C_VEL
LIN {X 0,Y 452.867,Z 466.054,A -85,B 0,C 180,E1 -8361.072,E2 -8361.072} C_VEL
LIN {X 0,Y 452.653,Z 471.533,A -85,B 0,C 180,E1 -8362.865,E2 -8362.865} C_VEL
LIN {X 0,Y 452.52,Z 475.675,A -85,B 0,C 180,E1 -8364.653,E2 -8364.653} C_VEL
LIN {X 0,Y 452.435,Z 478.578,A -85,B 0,C 180,E1 -8366.437,E2 -8366.437} C_VEL
LIN {X 0,Y 452.429,Z 480.31,A -85,B 0,C 180,E1 -8368.219,E2 -8368.219} C_VEL
LIN {X 0,Y 452.404,Z 480.903,A -85,B 0,C 180,E1 -8370,E2 -8370} C_VEL
LIN {X 0,Y 452.429,Z 480.308,A -85,B 0,C 180,E1 -8371.78,E2 -8371.78} C_VEL
LIN {X 0,Y 452.435,Z 478.573,A -85,B 0,C 180,E1 -8373.562,E2 -8373.562} C_VEL
LIN {X 0,Y 452.527,Z 475.673,A -85,B 0,C 180,E1 -8375.346,E2 -8375.346} C_VEL
LIN {X 0,Y 452.655,Z 471.538,A -85,B 0,C 180,E1 -8377.135,E2 -8377.135} C_VEL
LIN {X 0,Y 452.866,Z 466.055,A -85,B 0,C 180,E1 -8378.927,E2 -8378.927} C_VEL
LIN {X 0,Y 453.27,Z 459.078,A -85,B 0,C 180,E1 -8380.722,E2 -8380.722} C_VEL
LIN {X 0,Y 453.682,Z 451.608,A -85,B 0,C 180,E1 -8382.298,E2 -8382.298} C_VEL
LIN {X 0,Y 454.303,Z 442.601,A -85,B 0,C 180,E1 -8383.873,E2 -8383.873} C_VEL
LIN {X 0,Y 455.13,Z 431.777,A -85,B 0,C 180,E1 -8385.448,E2 -8385.448} C_VEL
LIN {X 0,Y 456.099,Z 419.608,A -85,B 0,C 180,E1 -8386.908,E2 -8386.908} C_VEL
LIN {X 0,Y 457.067,Z 407.193,A -85,B 0,C 180,E1 -8388.141,E2 -8388.141} C_VEL
LIN {X 0,Y 458.04,Z 393.455,A -85,B 0,C 180,E1 -8389.261,E2 -8389.261} C_VEL
LIN {X 0,Y 458.966,Z 379.964,A -85,B 0,C 180,E1 -8390.153,E2 -8390.153} C_VEL
LIN {X 0,Y 459.832,Z 364.961,A -85,B 0,C 180,E1 -8390.932,E2 -8390.932} C_VEL
LIN {X 0,Y 460.17,Z 354.799,A -85,B 0,C 180,E1 -8391.351,E2 -8391.351} C_VEL
LIN {X 0,Y 456.642,Z 339.826,A -85,B 0,C 180,E1 -8392.014,E2 -8392.014} C_VEL
LIN {X 0,Y 452.84,Z 326.16,A -85,B 0,C 180,E1 -8392.532,E2 -8392.532} C_VEL
LIN {X 0,Y 453.045,Z 320.091,A -85,B 0,C 180,E1 -8395.876,E2 -8395.876} C_VEL
LIN {X 0,Y 453.241,Z 315.048,A -85,B 0,C 180,E1 -8398.729,E2 -8398.729} C_VEL
LIN {X 0,Y 453.46,Z 309.736,A -85,B 0,C 180,E1 -8401.799,E2 -8401.799} C_VEL
LIN {X 0,Y 453.727,Z 304.652,A -85,B 0,C 180,E1 -8404.821,E2 -8404.821} C_VEL
LIN {X 0,Y 453.947,Z 299.75,A -85,B 0,C 180,E1 -8407.854,E2 -8407.854} C_VEL
LIN {X 0,Y 454.152,Z 295.362,A -85,B 0,C 180,E1 -8410.688,E2 -8410.688} C_VEL
LIN {X 0,Y 453.966,Z 291.522,A -85,B 0,C 180,E1 -8413.313,E2 -8413.313} C_VEL
LIN {X 0,Y 453.491,Z 288.625,A -85,B 0,C 180,E1 -8415.469,E2 -8415.469} C_VEL
LIN {X 0,Y 453.473,Z 288.626,A -85,B 0,C 180,E1 -8418.209,E2 -8418.209} C_VEL
LIN {X 0,Y 453.488,Z 288.623,A -85,B 0,C 180,E1 -8420.793,E2 -8420.793} C_VEL
LIN {X 0,Y 453.446,Z 288.629,A -85,B 0,C 180,E1 -8423.917,E2 -8423.917} C_VEL
LIN {X 0,Y 453.476,Z 288.626,A -85,B 0,C 180,E1 -8427.151,E2 -8427.151} C_VEL
LIN {X 0,Y 453.466,Z 288.627,A -85,B 0,C 180,E1 -8430.268,E2 -8430.268} C_VEL
LIN {X 0,Y 453.498,Z 288.621,A -85,B 0,C 180,E1 -8433.293,E2 -8433.293} C_VEL
LIN {X 0,Y 453.495,Z 288.62,A -85,B 0,C 180,E1 -8436.238,E2 -8436.238} C_VEL
LIN {X 0,Y 453.474,Z 288.623,A -85,B 0,C 180,E1 -8439.117,E2 -8439.117} C_VEL
LIN {X 0,Y 453.503,Z 288.62,A -85,B 0,C 180,E1 -8441.944,E2 -8441.944} C_VEL
LIN {X 0,Y 453.53,Z 288.618,A -85,B 0,C 180,E1 -8444.726,E2 -8444.726} C_VEL
LIN {X 0,Y 453.554,Z 288.612,A -85,B 0,C 180,E1 -8448.379,E2 -8448.379} C_VEL
LIN {X 0,Y 453.579,Z 288.61,A -85,B 0,C 180,E1 -8451.086,E2 -8451.086} C_VEL
LIN {X 0,Y 453.64,Z 288.604,A -85,B 0,C 180,E1 -8453.774,E2 -8453.774} C_VEL
LIN {X 0,Y 453.759,Z 288.585,A -85,B 0,C 180,E1 -8457.337,E2 -8457.337} C_VEL
LIN {X 0,Y 453.812,Z 288.584,A -85,B 0,C 180,E1 -8460,E2 -8460} C_VEL
LIN {X 0,Y 453.759,Z 288.588,A -85,B 0,C 180,E1 -8462.663,E2 -8462.663} C_VEL
LIN {X 0,Y 453.641,Z 288.606,A -85,B 0,C 180,E1 -8466.226,E2 -8466.226} C_VEL
LIN {X 0,Y 453.579,Z 288.609,A -85,B 0,C 180,E1 -8468.914,E2 -8468.914} C_VEL
LIN {X 0,Y 453.555,Z 288.614,A -85,B 0,C 180,E1 -8472.529,E2 -8472.529} C_VEL
LIN {X 0,Y 453.537,Z 288.615,A -85,B 0,C 180,E1 -8476.196,E2 -8476.196} C_VEL
LIN {X 0,Y 453.512,Z 288.618,A -85,B 0,C 180,E1 -8479.041,E2 -8479.041} C_VEL
LIN {X 0,Y 453.469,Z 288.624,A -85,B 0,C 180,E1 -8481.837,E2 -8481.837} C_VEL
LIN {X 0,Y 453.507,Z 288.62,A -85,B 0,C 180,E1 -8484.735,E2 -8484.735} C_VEL
LIN {X 0,Y 453.524,Z 288.616,A -85,B 0,C 180,E1 -8487.96,E2 -8487.96} C_VEL
LIN {X 0,Y 453.46,Z 288.622,A -85,B 0,C 180,E1 -8491.526,E2 -8491.526} C_VEL
LIN {X 0,Y 453.48,Z 288.621,A -85,B 0,C 180,E1 -8494.778,E2 -8494.778} C_VEL
LIN {X 0,Y 453.459,Z 288.628,A -85,B 0,C 180,E1 -8498.312,E2 -8498.312} C_VEL
LIN {X 0,Y 453.489,Z 288.622,A -85,B 0,C 180,E1 -8500.61,E2 -8500.61} C_VEL
LIN {X 0,Y 453.451,Z 288.627,A -85,B 0,C 180,E1 -8503.245,E2 -8503.245} C_VEL
LIN {X 0,Y 453.459,Z 288.629,A -85,B 0,C 180,E1 -8505.78,E2 -8505.78} C_VEL
LIN {X 0,Y 453.564,Z 289.557,A -85,B 0,C 180,E1 -8507.018,E2 -8507.018} C_VEL
LIN {X 0,Y 453.761,Z 292.561,A -85,B 0,C 180,E1 -8509.421,E2 -8509.421} C_VEL
LIN {X 0,Y 453.576,Z 296.229,A -85,B 0,C 180,E1 -8512.207,E2 -8512.207} C_VEL
LIN {X 0,Y 453.488,Z 300.332,A -85,B 0,C 180,E1 -8515.223,E2 -8515.223} C_VEL
LIN {X 0,Y 453.273,Z 304.985,A -85,B 0,C 180,E1 -8518.515,E2 -8518.515} C_VEL
LIN {X 0,Y 453.115,Z 308.996,A -85,B 0,C 180,E1 -8521.262,E2 -8521.262} C_VEL
LIN {X 0,Y 452.96,Z 313.509,A -85,B 0,C 180,E1 -8524.251,E2 -8524.251} C_VEL
LIN {X 0,Y 452.793,Z 318.577,A -85,B 0,C 180,E1 -8527.533,E2 -8527.533} C_VEL
LIN {X 0,Y 457.994,Z 336.516,A -85,B 0,C 180,E1 -8528.239,E2 -8528.239} C_VEL
LIN {X 0,Y 460.405,Z 346.665,A -85,B 0,C 180,E1 -8528.713,E2 -8528.713} C_VEL
LIN {X 0,Y 459.782,Z 361.091,A -85,B 0,C 180,E1 -8529.338,E2 -8529.338} C_VEL
LIN {X 0,Y 458.916,Z 374.476,A -85,B 0,C 180,E1 -8530.078,E2 -8530.078} C_VEL
LIN {X 0,Y 458.052,Z 387.431,A -85,B 0,C 180,E1 -8530.972,E2 -8530.972} C_VEL
LIN {X 0,Y 457.165,Z 399.501,A -85,B 0,C 180,E1 -8531.979,E2 -8531.979} C_VEL
LIN {X 0,Y 456.22,Z 411.751,A -85,B 0,C 180,E1 -8533.212,E2 -8533.212} C_VEL
LIN {X 0,Y 455.358,Z 422.589,A -85,B 0,C 180,E1 -8534.519,E2 -8534.519} C_VEL
LIN {X 0,Y 454.406,Z 426.678,A -85,B 0,C 180,E1 -8535.042,E2 -8535.042} C_VEL
LIN {X 0,Y 451.06,Z 433.05,A -85,B 0,C 180,E1 -8535.906,E2 -8535.906} C_VEL
LIN {X 0,Y 447.738,Z 439.051,A -85,B 0,C 180,E1 -8536.827,E2 -8536.827} C_VEL
LIN {X 0,Y 446.833,Z 442.421,A -85,B 0,C 180,E1 -8537.434,E2 -8537.434} C_VEL
LIN {X 0,Y 446.332,Z 450.288,A -85,B 0,C 180,E1 -8539.109,E2 -8539.109} C_VEL
LIN {X 0,Y 445.893,Z 457.265,A -85,B 0,C 180,E1 -8540.932,E2 -8540.932} C_VEL
LIN {X 0,Y 445.592,Z 462.75,A -85,B 0,C 180,E1 -8542.752,E2 -8542.752} C_VEL
LIN {X 0,Y 445.48,Z 466.892,A -85,B 0,C 180,E1 -8544.569,E2 -8544.569} C_VEL
LIN {X 0,Y 445.367,Z 469.805,A -85,B 0,C 180,E1 -8546.381,E2 -8546.381} C_VEL
LIN {X 0,Y 445.353,Z 471.559,A -85,B 0,C 180,E1 -8548.192,E2 -8548.192} C_VEL
LIN {X 0,Y 445.314,Z 472.173,A -85,B 0,C 180,E1 -8550,E2 -8550} C_VEL
LIN {X 0,Y 445.354,Z 471.609,A -85,B 0,C 180,E1 -8551.809,E2 -8551.809} C_VEL
LIN {X 0,Y 445.367,Z 469.922,A -85,B 0,C 180,E1 -8553.619,E2 -8553.619} C_VEL
LIN {X 0,Y 445.468,Z 467.071,A -85,B 0,C 180,E1 -8555.432,E2 -8555.432} C_VEL
LIN {X 0,Y 445.589,Z 462.992,A -85,B 0,C 180,E1 -8557.249,E2 -8557.249} C_VEL
LIN {X 0,Y 445.876,Z 457.582,A -85,B 0,C 180,E1 -8559.069,E2 -8559.069} C_VEL
LIN {X 0,Y 446.322,Z 450.691,A -85,B 0,C 180,E1 -8560.892,E2 -8560.892} C_VEL
LIN {X 0,Y 446.772,Z 443.285,A -85,B 0,C 180,E1 -8562.491,E2 -8562.491} C_VEL
LIN {X 0,Y 447.46,Z 434.358,A -85,B 0,C 180,E1 -8564.09,E2 -8564.09} C_VEL
LIN {X 0,Y 448.231,Z 425.261,A -85,B 0,C 180,E1 -8565.459,E2 -8565.459} C_VEL
LIN {X 0,Y 449.168,Z 414.53,A -85,B 0,C 180,E1 -8566.826,E2 -8566.826} C_VEL
LIN {X 0,Y 450.132,Z 402.726,A -85,B 0,C 180,E1 -8568.088,E2 -8568.088} C_VEL
LIN {X 0,Y 451.159,Z 390.033,A -85,B 0,C 180,E1 -8569.213,E2 -8569.213} C_VEL
LIN {X 0,Y 452.005,Z 377.689,A -85,B 0,C 180,E1 -8570.121,E2 -8570.121} C_VEL
LIN {X 0,Y 452.934,Z 364.447,A -85,B 0,C 180,E1 -8570.909,E2 -8570.909} C_VEL
LIN {X 0,Y 453.644,Z 350.338,A -85,B 0,C 180,E1 -8571.569,E2 -8571.569} C_VEL
LIN {X 0,Y 453.59,Z 347.077,A -85,B 0,C 180,E1 -8571.702,E2 -8571.702} C_VEL
LIN {X 0,Y 450.012,Z 333.02,A -85,B 0,C 180,E1 -8572.368,E2 -8572.368} C_VEL
LIN {X 0,Y 445.744,Z 318.667,A -85,B 0,C 180,E1 -8572.938,E2 -8572.938} C_VEL
LIN {X 0,Y 445.897,Z 313.767,A -85,B 0,C 180,E1 -8576.188,E2 -8576.188} C_VEL
LIN {X 0,Y 446.089,Z 309.269,A -85,B 0,C 180,E1 -8579.235,E2 -8579.235} C_VEL
LIN {X 0,Y 446.247,Z 304.783,A -85,B 0,C 180,E1 -8582.376,E2 -8582.376} C_VEL
LIN {X 0,Y 446.469,Z 300.272,A -85,B 0,C 180,E1 -8585.621,E2 -8585.621} C_VEL
LIN {X 0,Y 446.654,Z 295.748,A -85,B 0,C 180,E1 -8589.005,E2 -8589.005} C_VEL
LIN {X 0,Y 446.7,Z 292.73,A -85,B 0,C 180,E1 -8591.36,E2 -8591.36} C_VEL
LIN {X 0,Y 446.439,Z 289.721,A -85,B 0,C 180,E1 -8593.841,E2 -8593.841} C_VEL
LIN {X 0,Y 446.398,Z 289.508,A -85,B 0,C 180,E1 -8596.403,E2 -8596.403} C_VEL
LIN {X 0,Y 446.426,Z 289.502,A -85,B 0,C 180,E1 -8599.082,E2 -8599.082} C_VEL
LIN {X 0,Y 446.414,Z 289.507,A -85,B 0,C 180,E1 -8601.92,E2 -8601.92} C_VEL
LIN {X 0,Y 446.426,Z 289.503,A -85,B 0,C 180,E1 -8605.477,E2 -8605.477} C_VEL
LIN {X 0,Y 446.413,Z 289.503,A -85,B 0,C 180,E1 -8608.699,E2 -8608.699} C_VEL
LIN {X 0,Y 446.447,Z 289.498,A -85,B 0,C 180,E1 -8611.83,E2 -8611.83} C_VEL
LIN {X 0,Y 446.44,Z 289.499,A -85,B 0,C 180,E1 -8614.847,E2 -8614.847} C_VEL
LIN {X 0,Y 446.445,Z 289.497,A -85,B 0,C 180,E1 -8618.245,E2 -8618.245} C_VEL
LIN {X 0,Y 446.455,Z 289.499,A -85,B 0,C 180,E1 -8621.649,E2 -8621.649} C_VEL
LIN {X 0,Y 446.503,Z 289.491,A -85,B 0,C 180,E1 -8624.479,E2 -8624.479} C_VEL
LIN {X 0,Y 446.515,Z 289.491,A -85,B 0,C 180,E1 -8628.193,E2 -8628.193} C_VEL
LIN {X 0,Y 446.531,Z 289.491,A -85,B 0,C 180,E1 -8630.944,E2 -8630.944} C_VEL
LIN {X 0,Y 446.613,Z 289.479,A -85,B 0,C 180,E1 -8633.676,E2 -8633.676} C_VEL
LIN {X 0,Y 446.706,Z 289.467,A -85,B 0,C 180,E1 -8637.295,E2 -8637.295} C_VEL
LIN {X 0,Y 446.785,Z 289.459,A -85,B 0,C 180,E1 -8640,E2 -8640} C_VEL
LIN {X 0,Y 446.707,Z 289.467,A -85,B 0,C 180,E1 -8642.705,E2 -8642.705} C_VEL
LIN {X 0,Y 446.613,Z 289.48,A -85,B 0,C 180,E1 -8646.324,E2 -8646.324} C_VEL
LIN {X 0,Y 446.521,Z 289.489,A -85,B 0,C 180,E1 -8649.97,E2 -8649.97} C_VEL
LIN {X 0,Y 446.518,Z 289.49,A -85,B 0,C 180,E1 -8652.73,E2 -8652.73} C_VEL
LIN {X 0,Y 446.487,Z 289.494,A -85,B 0,C 180,E1 -8656.459,E2 -8656.459} C_VEL
LIN {X 0,Y 446.466,Z 289.496,A -85,B 0,C 180,E1 -8659.303,E2 -8659.303} C_VEL
LIN {X 0,Y 446.414,Z 289.502,A -85,B 0,C 180,E1 -8662.2,E2 -8662.2} C_VEL
LIN {X 0,Y 446.446,Z 289.498,A -85,B 0,C 180,E1 -8665.153,E2 -8665.153} C_VEL
LIN {X 0,Y 446.482,Z 289.496,A -85,B 0,C 180,E1 -8668.179,E2 -8668.179} C_VEL
LIN {X 0,Y 446.415,Z 289.507,A -85,B 0,C 180,E1 -8671.775,E2 -8671.775} C_VEL
LIN {X 0,Y 446.425,Z 289.506,A -85,B 0,C 180,E1 -8674.523,E2 -8674.523} C_VEL
LIN {X 0,Y 446.41,Z 289.509,A -85,B 0,C 180,E1 -8678.079,E2 -8678.079} C_VEL
LIN {X 0,Y 446.42,Z 289.505,A -85,B 0,C 180,E1 -8680.917,E2 -8680.917} C_VEL
LIN {X 0,Y 446.455,Z 289.592,A -85,B 0,C 180,E1 -8684.385,E2 -8684.385} C_VEL
LIN {X 0,Y 446.892,Z 292.217,A -85,B 0,C 180,E1 -8686.337,E2 -8686.337} C_VEL
LIN {X 0,Y 447.13,Z 295.989,A -85,B 0,C 180,E1 -8688.979,E2 -8688.979} C_VEL
LIN {X 0,Y 446.918,Z 300.831,A -85,B 0,C 180,E1 -8692.172,E2 -8692.172} C_VEL
LIN {X 0,Y 446.663,Z 306.095,A -85,B 0,C 180,E1 -8695.498,E2 -8695.498} C_VEL
LIN {X 0,Y 446.383,Z 311.396,A -85,B 0,C 180,E1 -8698.697,E2 -8698.697} C_VEL
LIN {X 0,Y 446.134,Z 316.681,A -85,B 0,C 180,E1 -8701.797,E2 -8701.797} C_VEL
LIN {X 0,Y 445.917,Z 321.99,A -85,B 0,C 180,E1 -8704.815,E2 -8704.815} C_VEL
LIN {X 0,Y 445.783,Z 326.094,A -85,B 0,C 180,E1 -8707.102,E2 -8707.102} C_VEL
LIN {X 0,Y 450.783,Z 344.072,A -85,B 0,C 180,E1 -8707.803,E2 -8707.803} C_VEL
LIN {X 0,Y 453.591,Z 357.264,A -85,B 0,C 180,E1 -8708.421,E2 -8708.421} C_VEL
LIN {X 0,Y 452.87,Z 371.821,A -85,B 0,C 180,E1 -8709.088,E2 -8709.088} C_VEL
LIN {X 0,Y 451.904,Z 385.272,A -85,B 0,C 180,E1 -8709.874,E2 -8709.874} C_VEL
LIN {X 0,Y 450.988,Z 397.774,A -85,B 0,C 180,E1 -8710.78,E2 -8710.78} C_VEL
LIN {X 0,Y 449.967,Z 410.808,A -85,B 0,C 180,E1 -8711.927,E2 -8711.927} C_VEL
LIN {X 0,Y 449.036,Z 422.515,A -85,B 0,C 180,E1 -8713.169,E2 -8713.169} C_VEL
LIN {X 0,Y 448.099,Z 433.347,A -85,B 0,C 180,E1 -8714.536,E2 -8714.536} C_VEL
LIN {X 0,Y 447.238,Z 443.891,A -85,B 0,C 180,E1 -8716.134,E2 -8716.134} C_VEL
LIN {X 0,Y 446.586,Z 452.665,A -85,B 0,C 180,E1 -8717.734,E2 -8717.734} C_VEL
LIN {X 0,Y 446.267,Z 459.016,A -85,B 0,C 180,E1 -8719.107,E2 -8719.107} C_VEL
LIN {X 0,Y 445.804,Z 465.986,A -85,B 0,C 180,E1 -8720.929,E2 -8720.929} C_VEL
LIN {X 0,Y 445.578,Z 471.465,A -85,B 0,C 180,E1 -8722.751,E2 -8722.751} C_VEL
LIN {X 0,Y 445.439,Z 475.606,A -85,B 0,C 180,E1 -8724.568,E2 -8724.568} C_VEL
LIN {X 0,Y 445.334,Z 478.509,A -85,B 0,C 180,E1 -8726.38,E2 -8726.38} C_VEL
LIN {X 0,Y 445.349,Z 480.241,A -85,B 0,C 180,E1 -8728.191,E2 -8728.191} C_VEL
LIN {X 0,Y 445.313,Z 480.835,A -85,B 0,C 180,E1 -8730,E2 -8730} C_VEL
LIN {X 0,Y 445.348,Z 480.239,A -85,B 0,C 180,E1 -8731.808,E2 -8731.808} C_VEL
LIN {X 0,Y 445.334,Z 478.504,A -85,B 0,C 180,E1 -8733.619,E2 -8733.619} C_VEL
LIN {X 0,Y 445.449,Z 475.604,A -85,B 0,C 180,E1 -8735.432,E2 -8735.432} C_VEL
LIN {X 0,Y 445.579,Z 471.468,A -85,B 0,C 180,E1 -8737.249,E2 -8737.249} C_VEL
LIN {X 0,Y 445.803,Z 465.985,A -85,B 0,C 180,E1 -8739.07,E2 -8739.07} C_VEL
LIN {X 0,Y 446.264,Z 459.007,A -85,B 0,C 180,E1 -8740.893,E2 -8740.893} C_VEL
LIN {X 0,Y 446.694,Z 451.244,A -85,B 0,C 180,E1 -8742.551,E2 -8742.551} C_VEL
LIN {X 0,Y 447.372,Z 442.53,A -85,B 0,C 180,E1 -8744.092,E2 -8744.092} C_VEL
LIN {X 0,Y 448.242,Z 431.706,A -85,B 0,C 180,E1 -8745.691,E2 -8745.691} C_VEL
LIN {X 0,Y 449.269,Z 419.536,A -85,B 0,C 180,E1 -8747.173,E2 -8747.173} C_VEL
LIN {X 0,Y 450.295,Z 407.121,A -85,B 0,C 180,E1 -8748.424,E2 -8748.424} C_VEL
LIN {X 0,Y 451.304,Z 393.382,A -85,B 0,C 180,E1 -8749.56,E2 -8749.56} C_VEL
LIN {X 0,Y 452.301,Z 379.89,A -85,B 0,C 180,E1 -8750.463,E2 -8750.463} C_VEL
LIN {X 0,Y 453.157,Z 365.822,A -85,B 0,C 180,E1 -8751.211,E2 -8751.211} C_VEL
LIN {X 0,Y 453.476,Z 356.163,A -85,B 0,C 180,E1 -8751.626,E2 -8751.626} C_VEL
LIN {X 0,Y 450.293,Z 342.255,A -85,B 0,C 180,E1 -8752.275,E2 -8752.275} C_VEL
LIN {X 0,Y 445.774,Z 326.116,A -85,B 0,C 180,E1 -8752.896,E2 -8752.896} C_VEL
LIN {X 0,Y 445.987,Z 320.263,A -85,B 0,C 180,E1 -8756.182,E2 -8756.182} C_VEL
LIN {X 0,Y 446.209,Z 314.989,A -85,B 0,C 180,E1 -8759.226,E2 -8759.226} C_VEL
LIN {X 0,Y 446.457,Z 309.682,A -85,B 0,C 180,E1 -8762.358,E2 -8762.358} C_VEL
LIN {X 0,Y 446.735,Z 304.365,A -85,B 0,C 180,E1 -8765.596,E2 -8765.596} C_VEL
LIN {X 0,Y 447.022,Z 299.068,A -85,B 0,C 180,E1 -8768.966,E2 -8768.966} C_VEL
LIN {X 0,Y 447.117,Z 295.548,A -85,B 0,C 180,E1 -8771.312,E2 -8771.312} C_VEL
LIN {X 0,Y 446.87,Z 292.026,A -85,B 0,C 180,E1 -8773.787,E2 -8773.787} C_VEL
LIN {X 0,Y 446.433,Z 289.504,A -85,B 0,C 180,E1 -8775.749,E2 -8775.749} C_VEL
LIN {X 0,Y 446.421,Z 289.505,A -85,B 0,C 180,E1 -8779.082,E2 -8779.082} C_VEL
LIN {X 0,Y 446.409,Z 289.507,A -85,B 0,C 180,E1 -8781.92,E2 -8781.92} C_VEL
LIN {X 0,Y 446.421,Z 289.505,A -85,B 0,C 180,E1 -8785.476,E2 -8785.476} C_VEL
LIN {X 0,Y 446.409,Z 289.507,A -85,B 0,C 180,E1 -8788.699,E2 -8788.699} C_VEL
LIN {X 0,Y 446.477,Z 289.497,A -85,B 0,C 180,E1 -8791.821,E2 -8791.821} C_VEL
LIN {X 0,Y 446.449,Z 289.498,A -85,B 0,C 180,E1 -8794.847,E2 -8794.847} C_VEL
LIN {X 0,Y 446.44,Z 289.5,A -85,B 0,C 180,E1 -8798.245,E2 -8798.245} C_VEL
LIN {X 0,Y 446.449,Z 289.501,A -85,B 0,C 180,E1 -8801.649,E2 -8801.649} C_VEL
LIN {X 0,Y 446.498,Z 289.494,A -85,B 0,C 180,E1 -8804.48,E2 -8804.48} C_VEL
LIN {X 0,Y 446.511,Z 289.49,A -85,B 0,C 180,E1 -8808.193,E2 -8808.193} C_VEL
LIN {X 0,Y 446.527,Z 289.489,A -85,B 0,C 180,E1 -8810.945,E2 -8810.945} C_VEL
LIN {X 0,Y 446.609,Z 289.48,A -85,B 0,C 180,E1 -8813.676,E2 -8813.676} C_VEL
LIN {X 0,Y 446.703,Z 289.464,A -85,B 0,C 180,E1 -8817.295,E2 -8817.295} C_VEL
LIN {X 0,Y 446.781,Z 289.46,A -85,B 0,C 180,E1 -8820,E2 -8820} C_VEL
LIN {X 0,Y 446.703,Z 289.467,A -85,B 0,C 180,E1 -8822.705,E2 -8822.705} C_VEL
LIN {X 0,Y 446.594,Z 289.481,A -85,B 0,C 180,E1 -8826.473,E2 -8826.473} C_VEL
LIN {X 0,Y 446.517,Z 289.489,A -85,B 0,C 180,E1 -8829.97,E2 -8829.97} C_VEL
LIN {X 0,Y 446.513,Z 289.49,A -85,B 0,C 180,E1 -8832.73,E2 -8832.73} C_VEL
LIN {X 0,Y 446.482,Z 289.495,A -85,B 0,C 180,E1 -8836.459,E2 -8836.459} C_VEL
LIN {X 0,Y 446.462,Z 289.497,A -85,B 0,C 180,E1 -8839.304,E2 -8839.304} C_VEL
LIN {X 0,Y 446.41,Z 289.502,A -85,B 0,C 180,E1 -8842.2,E2 -8842.2} C_VEL
LIN {X 0,Y 446.45,Z 289.497,A -85,B 0,C 180,E1 -8845.153,E2 -8845.153} C_VEL
LIN {X 0,Y 446.478,Z 289.492,A -85,B 0,C 180,E1 -8848.179,E2 -8848.179} C_VEL
LIN {X 0,Y 446.413,Z 289.501,A -85,B 0,C 180,E1 -8851.776,E2 -8851.776} C_VEL
LIN {X 0,Y 446.422,Z 289.499,A -85,B 0,C 180,E1 -8854.524,E2 -8854.524} C_VEL
LIN {X 0,Y 446.41,Z 289.505,A -85,B 0,C 180,E1 -8858.08,E2 -8858.08} C_VEL
LIN {X 0,Y 446.422,Z 289.504,A -85,B 0,C 180,E1 -8860.918,E2 -8860.918} C_VEL
LIN {X 0,Y 446.397,Z 289.505,A -85,B 0,C 180,E1 -8863.847,E2 -8863.847} C_VEL
LIN {X 0,Y 446.406,Z 289.6,A -85,B 0,C 180,E1 -8866.156,E2 -8866.156} C_VEL
LIN {X 0,Y 446.7,Z 293.103,A -85,B 0,C 180,E1 -8869.042,E2 -8869.042} C_VEL
LIN {X 0,Y 446.567,Z 296.785,A -85,B 0,C 180,E1 -8871.896,E2 -8871.896} C_VEL
LIN {X 0,Y 446.443,Z 300.856,A -85,B 0,C 180,E1 -8874.945,E2 -8874.945} C_VEL
LIN {X 0,Y 446.222,Z 305.472,A -85,B 0,C 180,E1 -8878.266,E2 -8878.266} C_VEL
LIN {X 0,Y 446.081,Z 309.055,A -85,B 0,C 180,E1 -8880.765,E2 -8880.765} C_VEL
LIN {X 0,Y 445.924,Z 313.764,A -85,B 0,C 180,E1 -8883.942,E2 -8883.942} C_VEL
LIN {X 0,Y 445.731,Z 318.665,A -85,B 0,C 180,E1 -8887.168,E2 -8887.168} C_VEL
LIN {X 0,Y 450.545,Z 334.875,A -85,B 0,C 180,E1 -8887.804,E2 -8887.804} C_VEL
LIN {X 0,Y 453.731,Z 347.925,A -85,B 0,C 180,E1 -8888.431,E2 -8888.431} C_VEL
LIN {X 0,Y 453.009,Z 362.707,A -85,B 0,C 180,E1 -8889.096,E2 -8889.096} C_VEL
LIN {X 0,Y 452.081,Z 376.316,A -85,B 0,C 180,E1 -8889.883,E2 -8889.883} C_VEL
LIN {X 0,Y 451.08,Z 390.356,A -85,B 0,C 180,E1 -8890.902,E2 -8890.902} C_VEL
LIN {X 0,Y 450.121,Z 402.95,A -85,B 0,C 180,E1 -8892.026,E2 -8892.026} C_VEL
LIN {X 0,Y 449.213,Z 413.775,A -85,B 0,C 180,E1 -8893.176,E2 -8893.176} C_VEL
LIN {X 0,Y 448.286,Z 424.625,A -85,B 0,C 180,E1 -8894.543,E2 -8894.543} C_VEL
LIN {X 0,Y 447.534,Z 433.828,A -85,B 0,C 180,E1 -8895.913,E2 -8895.913} C_VEL
LIN {X 0,Y 446.833,Z 442.421,A -85,B 0,C 180,E1 -8897.434,E2 -8897.434} C_VEL
LIN {X 0,Y 445.965,Z 445.692,A -85,B 0,C 180,E1 -8898.055,E2 -8898.055} C_VEL
LIN {X 0,Y 442.806,Z 450.689,A -85,B 0,C 180,E1 -8899.082,E2 -8899.082} C_VEL
LIN {X 0,Y 439.665,Z 455.145,A -85,B 0,C 180,E1 -8900.161,E2 -8900.161} C_VEL
LIN {X 0,Y 438.843,Z 457.571,A -85,B 0,C 180,E1 -8900.858,E2 -8900.858} C_VEL
LIN {X 0,Y 438.518,Z 462.82,A -85,B 0,C 180,E1 -8902.634,E2 -8902.634} C_VEL
LIN {X 0,Y 438.402,Z 466.962,A -85,B 0,C 180,E1 -8904.481,E2 -8904.481} C_VEL
LIN {X 0,Y 438.268,Z 469.875,A -85,B 0,C 180,E1 -8906.323,E2 -8906.323} C_VEL
LIN {X 0,Y 438.276,Z 471.628,A -85,B 0,C 180,E1 -8908.163,E2 -8908.163} C_VEL
LIN {X 0,Y 438.227,Z 472.242,A -85,B 0,C 180,E1 -8910,E2 -8910} C_VEL
LIN {X 0,Y 438.276,Z 471.677,A -85,B 0,C 180,E1 -8911.838,E2 -8911.838} C_VEL
LIN {X 0,Y 438.268,Z 469.99,A -85,B 0,C 180,E1 -8913.678,E2 -8913.678} C_VEL
LIN {X 0,Y 438.39,Z 467.14,A -85,B 0,C 180,E1 -8915.52,E2 -8915.52} C_VEL
LIN {X 0,Y 438.516,Z 463.06,A -85,B 0,C 180,E1 -8917.367,E2 -8917.367} C_VEL
LIN {X 0,Y 438.821,Z 457.65,A -85,B 0,C 180,E1 -8919.216,E2 -8919.216} C_VEL
LIN {X 0,Y 439.337,Z 450.758,A -85,B 0,C 180,E1 -8921.067,E2 -8921.067} C_VEL
LIN {X 0,Y 439.814,Z 443.145,A -85,B 0,C 180,E1 -8922.735,E2 -8922.735} C_VEL
LIN {X 0,Y 440.533,Z 434.425,A -85,B 0,C 180,E1 -8924.317,E2 -8924.317} C_VEL
LIN {X 0,Y 441.343,Z 425.327,A -85,B 0,C 180,E1 -8925.707,E2 -8925.707} C_VEL
LIN {X 0,Y 442.34,Z 414.596,A -85,B 0,C 180,E1 -8927.094,E2 -8927.094} C_VEL
LIN {X 0,Y 443.35,Z 402.878,A -85,B 0,C 180,E1 -8928.365,E2 -8928.365} C_VEL
LIN {X 0,Y 444.437,Z 390.097,A -85,B 0,C 180,E1 -8929.515,E2 -8929.515} C_VEL
LIN {X 0,Y 445.324,Z 377.752,A -85,B 0,C 180,E1 -8930.437,E2 -8930.437} C_VEL
LIN {X 0,Y 446.29,Z 364.507,A -85,B 0,C 180,E1 -8931.235,E2 -8931.235} C_VEL
LIN {X 0,Y 447.075,Z 350.316,A -85,B 0,C 180,E1 -8931.906,E2 -8931.906} C_VEL
LIN {X 0,Y 446.558,Z 346.736,A -85,B 0,C 180,E1 -8932.077,E2 -8932.077} C_VEL
LIN {X 0,Y 442.781,Z 332.368,A -85,B 0,C 180,E1 -8932.772,E2 -8932.772} C_VEL
LIN {X 0,Y 438.709,Z 318.728,A -85,B 0,C 180,E1 -8933.333,E2 -8933.333} C_VEL
LIN {X 0,Y 438.845,Z 313.825,A -85,B 0,C 180,E1 -8936.642,E2 -8936.642} C_VEL
LIN {X 0,Y 439.085,Z 309.334,A -85,B 0,C 180,E1 -8939.748,E2 -8939.748} C_VEL
LIN {X 0,Y 439.245,Z 304.836,A -85,B 0,C 180,E1 -8942.957,E2 -8942.957} C_VEL
LIN {X 0,Y 439.431,Z 301.56,A -85,B 0,C 180,E1 -8945.347,E2 -8945.347} C_VEL
LIN {X 0,Y 439.591,Z 297.299,A -85,B 0,C 180,E1 -8948.573,E2 -8948.573} C_VEL
LIN {X 0,Y 439.678,Z 293.839,A -85,B 0,C 180,E1 -8951.3,E2 -8951.3} C_VEL
LIN {X 0,Y 439.418,Z 290.652,A -85,B 0,C 180,E1 -8953.968,E2 -8953.968} C_VEL
LIN {X 0,Y 439.366,Z 290.386,A -85,B 0,C 180,E1 -8956.038,E2 -8956.038} C_VEL
LIN {X 0,Y 439.38,Z 290.38,A -85,B 0,C 180,E1 -8959.019,E2 -8959.019} C_VEL
LIN {X 0,Y 439.376,Z 290.382,A -85,B 0,C 180,E1 -8961.607,E2 -8961.607} C_VEL
LIN {X 0,Y 439.397,Z 290.381,A -85,B 0,C 180,E1 -8964.844,E2 -8964.844} C_VEL
LIN {X 0,Y 439.37,Z 290.383,A -85,B 0,C 180,E1 -8968.139,E2 -8968.139} C_VEL
LIN {X 0,Y 439.406,Z 290.375,A -85,B 0,C 180,E1 -8971.604,E2 -8971.604} C_VEL
LIN {X 0,Y 439.377,Z 290.38,A -85,B 0,C 180,E1 -8974.413,E2 -8974.413} C_VEL
LIN {X 0,Y 439.361,Z 290.381,A -85,B 0,C 180,E1 -8977.424,E2 -8977.424} C_VEL
LIN {X 0,Y 439.439,Z 290.37,A -85,B 0,C 180,E1 -8980.663,E2 -8980.663} C_VEL
LIN {X 0,Y 439.459,Z 290.367,A -85,B 0,C 180,E1 -8984.224,E2 -8984.224} C_VEL
LIN {X 0,Y 439.481,Z 290.369,A -85,B 0,C 180,E1 -8988.001,E2 -8988.001} C_VEL
LIN {X 0,Y 439.494,Z 290.368,A -85,B 0,C 180,E1 -8990.798,E2 -8990.798} C_VEL
LIN {X 0,Y 439.564,Z 290.356,A -85,B 0,C 180,E1 -8993.574,E2 -8993.574} C_VEL
LIN {X 0,Y 439.43,Z 290.375,A -85,B 0,C 180,E1 -8995.413,E2 -8995.413} C_VEL
LIN {X 0,Y 439.653,Z 290.346,A -85,B 0,C 180,E1 -8997.251,E2 -8997.251} C_VEL
LIN {X 0,Y 439.754,Z 290.335,A -85,B 0,C 180,E1 -9000,E2 -9000} C_VEL
LIN {X 0,Y 439.653,Z 290.346,A -85,B 0,C 180,E1 -9002.749,E2 -9002.749} C_VEL
LIN {X 0,Y 439.564,Z 290.357,A -85,B 0,C 180,E1 -9006.426,E2 -9006.426} C_VEL
LIN {X 0,Y 439.494,Z 290.368,A -85,B 0,C 180,E1 -9009.202,E2 -9009.202} C_VEL
LIN {X 0,Y 439.462,Z 290.369,A -85,B 0,C 180,E1 -9012.938,E2 -9012.938} C_VEL
LIN {X 0,Y 439.444,Z 290.371,A -85,B 0,C 180,E1 -9016.349,E2 -9016.349} C_VEL
LIN {X 0,Y 439.399,Z 290.378,A -85,B 0,C 180,E1 -9019.626,E2 -9019.626} C_VEL
LIN {X 0,Y 439.361,Z 290.382,A -85,B 0,C 180,E1 -9022.576,E2 -9022.576} C_VEL
LIN {X 0,Y 439.397,Z 290.377,A -85,B 0,C 180,E1 -9025.585,E2 -9025.585} C_VEL
LIN {X 0,Y 439.414,Z 290.377,A -85,B 0,C 180,E1 -9028.674,E2 -9028.674} C_VEL
LIN {X 0,Y 439.366,Z 290.387,A -85,B 0,C 180,E1 -9032.03,E2 -9032.03} C_VEL
LIN {X 0,Y 439.391,Z 290.385,A -85,B 0,C 180,E1 -9035.34,E2 -9035.34} C_VEL
LIN {X 0,Y 439.367,Z 290.385,A -85,B 0,C 180,E1 -9038.596,E2 -9038.596} C_VEL
LIN {X 0,Y 439.379,Z 290.382,A -85,B 0,C 180,E1 -9041.256,E2 -9041.256} C_VEL
LIN {X 0,Y 439.382,Z 290.434,A -85,B 0,C 180,E1 -9044.095,E2 -9044.095} C_VEL
LIN {X 0,Y 439.908,Z 293.764,A -85,B 0,C 180,E1 -9046.61,E2 -9046.61} C_VEL
LIN {X 0,Y 440.107,Z 297.278,A -85,B 0,C 180,E1 -9049.102,E2 -9049.102} C_VEL
LIN {X 0,Y 439.954,Z 300.854,A -85,B 0,C 180,E1 -9051.512,E2 -9051.512} C_VEL
LIN {X 0,Y 439.668,Z 306.051,A -85,B 0,C 180,E1 -9054.869,E2 -9054.869} C_VEL
LIN {X 0,Y 439.374,Z 311.332,A -85,B 0,C 180,E1 -9058.14,E2 -9058.14} C_VEL
LIN {X 0,Y 439.209,Z 314.866,A -85,B 0,C 180,E1 -9060.261,E2 -9060.261} C_VEL
LIN {X 0,Y 438.925,Z 320.774,A -85,B 0,C 180,E1 -9063.723,E2 -9063.723} C_VEL
LIN {X 0,Y 438.748,Z 326.033,A -85,B 0,C 180,E1 -9066.718,E2 -9066.718} C_VEL
LIN {X 0,Y 443.642,Z 343.425,A -85,B 0,C 180,E1 -9067.407,E2 -9067.407} C_VEL
LIN {X 0,Y 446.897,Z 357.708,A -85,B 0,C 180,E1 -9068.101,E2 -9068.101} C_VEL
LIN {X 0,Y 446.163,Z 372.877,A -85,B 0,C 180,E1 -9068.819,E2 -9068.819} C_VEL
LIN {X 0,Y 445.108,Z 386.973,A -85,B 0,C 180,E1 -9069.674,E2 -9069.674} C_VEL
LIN {X 0,Y 444.04,Z 400.56,A -85,B 0,C 180,E1 -9070.707,E2 -9070.707} C_VEL
LIN {X 0,Y 442.899,Z 414.124,A -85,B 0,C 180,E1 -9071.976,E2 -9071.976} C_VEL
LIN {X 0,Y 441.831,Z 426.311,A -85,B 0,C 180,E1 -9073.362,E2 -9073.362} C_VEL
LIN {X 0,Y 440.917,Z 436.538,A -85,B 0,C 180,E1 -9074.752,E2 -9074.752} C_VEL
LIN {X 0,Y 440.083,Z 446.535,A -85,B 0,C 180,E1 -9076.376,E2 -9076.376} C_VEL
LIN {X 0,Y 439.448,Z 454.835,A -85,B 0,C 180,E1 -9078,E2 -9078} C_VEL
LIN {X 0,Y 439.045,Z 460.818,A -85,B 0,C 180,E1 -9079.392,E2 -9079.392} C_VEL
LIN {X 0,Y 438.678,Z 467.405,A -85,B 0,C 180,E1 -9081.245,E2 -9081.245} C_VEL
LIN {X 0,Y 438.439,Z 472.557,A -85,B 0,C 180,E1 -9083.095,E2 -9083.095} C_VEL
LIN {X 0,Y 438.342,Z 475.537,A -85,B 0,C 180,E1 -9084.479,E2 -9084.479} C_VEL
LIN {X 0,Y 438.237,Z 478.44,A -85,B 0,C 180,E1 -9086.322,E2 -9086.322} C_VEL
LIN {X 0,Y 438.27,Z 480.172,A -85,B 0,C 180,E1 -9088.162,E2 -9088.162} C_VEL
LIN {X 0,Y 438.225,Z 480.766,A -85,B 0,C 180,E1 -9090,E2 -9090} C_VEL
LIN {X 0,Y 438.27,Z 480.17,A -85,B 0,C 180,E1 -9091.837,E2 -9091.837} C_VEL
LIN {X 0,Y 438.237,Z 478.434,A -85,B 0,C 180,E1 -9093.678,E2 -9093.678} C_VEL
LIN {X 0,Y 438.354,Z 475.534,A -85,B 0,C 180,E1 -9095.52,E2 -9095.52} C_VEL
LIN {X 0,Y 438.5,Z 471.398,A -85,B 0,C 180,E1 -9097.366,E2 -9097.366} C_VEL
LIN {X 0,Y 438.728,Z 465.914,A -85,B 0,C 180,E1 -9099.217,E2 -9099.217} C_VEL
LIN {X 0,Y 439.232,Z 458.936,A -85,B 0,C 180,E1 -9101.069,E2 -9101.069} C_VEL
LIN {X 0,Y 439.766,Z 450.249,A -85,B 0,C 180,E1 -9102.928,E2 -9102.928} C_VEL
LIN {X 0,Y 440.546,Z 441.02,A -85,B 0,C 180,E1 -9104.551,E2 -9104.551} C_VEL
LIN {X 0,Y 441.346,Z 431.634,A -85,B 0,C 180,E1 -9105.943,E2 -9105.943} C_VEL
LIN {X 0,Y 442.342,Z 420.483,A -85,B 0,C 180,E1 -9107.331,E2 -9107.331} C_VEL
LIN {X 0,Y 443.416,Z 408.265,A -85,B 0,C 180,E1 -9108.6,E2 -9108.6} C_VEL
LIN {X 0,Y 444.467,Z 394.827,A -85,B 0,C 180,E1 -9109.753,E2 -9109.753} C_VEL
LIN {X 0,Y 445.5,Z 381.63,A -85,B 0,C 180,E1 -9110.669,E2 -9110.669} C_VEL
LIN {X 0,Y 446.458,Z 367.482,A -85,B 0,C 180,E1 -9111.453,E2 -9111.453} C_VEL
LIN {X 0,Y 446.741,Z 357.197,A -85,B 0,C 180,E1 -9111.924,E2 -9111.924} C_VEL
LIN {X 0,Y 443.833,Z 344.31,A -85,B 0,C 180,E1 -9112.55,E2 -9112.55} C_VEL
LIN {X 0,Y 439.455,Z 328.815,A -85,B 0,C 180,E1 -9113.177,E2 -9113.177} C_VEL
LIN {X 0,Y 438.742,Z 326.051,A -85,B 0,C 180,E1 -9113.28,E2 -9113.28} C_VEL
LIN {X 0,Y 438.937,Z 320.2,A -85,B 0,C 180,E1 -9116.635,E2 -9116.635} C_VEL
LIN {X 0,Y 439.208,Z 314.929,A -85,B 0,C 180,E1 -9119.738,E2 -9119.738} C_VEL
LIN {X 0,Y 439.461,Z 309.627,A -85,B 0,C 180,E1 -9122.938,E2 -9122.938} C_VEL
LIN {X 0,Y 439.763,Z 304.314,A -85,B 0,C 180,E1 -9126.249,E2 -9126.249} C_VEL
LIN {X 0,Y 440.035,Z 299.023,A -85,B 0,C 180,E1 -9129.706,E2 -9129.706} C_VEL
LIN {X 0,Y 440.062,Z 295.505,A -85,B 0,C 180,E1 -9132.124,E2 -9132.124} C_VEL
LIN {X 0,Y 439.694,Z 291.989,A -85,B 0,C 180,E1 -9134.69,E2 -9134.69} C_VEL
LIN {X 0,Y 439.379,Z 290.382,A -85,B 0,C 180,E1 -9136.035,E2 -9136.035} C_VEL
LIN {X 0,Y 439.374,Z 290.383,A -85,B 0,C 180,E1 -9139.019,E2 -9139.019} C_VEL
LIN {X 0,Y 439.368,Z 290.384,A -85,B 0,C 180,E1 -9141.607,E2 -9141.607} C_VEL
LIN {X 0,Y 439.391,Z 290.383,A -85,B 0,C 180,E1 -9144.843,E2 -9144.843} C_VEL
LIN {X 0,Y 439.366,Z 290.386,A -85,B 0,C 180,E1 -9148.139,E2 -9148.139} C_VEL
LIN {X 0,Y 439.425,Z 290.375,A -85,B 0,C 180,E1 -9151.598,E2 -9151.598} C_VEL
LIN {X 0,Y 439.397,Z 290.377,A -85,B 0,C 180,E1 -9154.415,E2 -9154.415} C_VEL
LIN {X 0,Y 439.357,Z 290.382,A -85,B 0,C 180,E1 -9157.424,E2 -9157.424} C_VEL
LIN {X 0,Y 439.433,Z 290.372,A -85,B 0,C 180,E1 -9160.663,E2 -9160.663} C_VEL
LIN {X 0,Y 439.454,Z 290.37,A -85,B 0,C 180,E1 -9164.224,E2 -9164.224} C_VEL
LIN {X 0,Y 439.476,Z 290.367,A -85,B 0,C 180,E1 -9168.001,E2 -9168.001} C_VEL
LIN {X 0,Y 439.49,Z 290.366,A -85,B 0,C 180,E1 -9170.798,E2 -9170.798} C_VEL
LIN {X 0,Y 439.559,Z 290.358,A -85,B 0,C 180,E1 -9173.574,E2 -9173.574} C_VEL
LIN {X 0,Y 439.429,Z 290.375,A -85,B 0,C 180,E1 -9175.413,E2 -9175.413} C_VEL
LIN {X 0,Y 439.65,Z 290.343,A -85,B 0,C 180,E1 -9177.251,E2 -9177.251} C_VEL
LIN {X 0,Y 439.751,Z 290.336,A -85,B 0,C 180,E1 -9180,E2 -9180} C_VEL
LIN {X 0,Y 439.65,Z 290.346,A -85,B 0,C 180,E1 -9182.749,E2 -9182.749} C_VEL
LIN {X 0,Y 439.556,Z 290.358,A -85,B 0,C 180,E1 -9186.462,E2 -9186.462} C_VEL
LIN {X 0,Y 439.489,Z 290.367,A -85,B 0,C 180,E1 -9189.202,E2 -9189.202} C_VEL
LIN {X 0,Y 439.457,Z 290.369,A -85,B 0,C 180,E1 -9192.938,E2 -9192.938} C_VEL
LIN {X 0,Y 439.439,Z 290.372,A -85,B 0,C 180,E1 -9196.349,E2 -9196.349} C_VEL
LIN {X 0,Y 439.395,Z 290.379,A -85,B 0,C 180,E1 -9199.627,E2 -9199.627} C_VEL
LIN {X 0,Y 439.357,Z 290.382,A -85,B 0,C 180,E1 -9202.576,E2 -9202.576} C_VEL
LIN {X 0,Y 439.398,Z 290.376,A -85,B 0,C 180,E1 -9205.585,E2 -9205.585} C_VEL
LIN {X 0,Y 439.41,Z 290.374,A -85,B 0,C 180,E1 -9208.674,E2 -9208.674} C_VEL
LIN {X 0,Y 439.364,Z 290.381,A -85,B 0,C 180,E1 -9212.031,E2 -9212.031} C_VEL
LIN {X 0,Y 439.388,Z 290.379,A -85,B 0,C 180,E1 -9215.341,E2 -9215.341} C_VEL
LIN {X 0,Y 439.379,Z 290.381,A -85,B 0,C 180,E1 -9218.595,E2 -9218.595} C_VEL
LIN {X 0,Y 439.383,Z 290.381,A -85,B 0,C 180,E1 -9221.257,E2 -9221.257} C_VEL
LIN {X 0,Y 439.396,Z 290.378,A -85,B 0,C 180,E1 -9224.73,E2 -9224.73} C_VEL
LIN {X 0,Y 439.39,Z 290.538,A -85,B 0,C 180,E1 -9226.036,E2 -9226.036} C_VEL
LIN {X 0,Y 439.691,Z 294.145,A -85,B 0,C 180,E1 -9229.056,E2 -9229.056} C_VEL
LIN {X 0,Y 439.572,Z 297.338,A -85,B 0,C 180,E1 -9231.575,E2 -9231.575} C_VEL
LIN {X 0,Y 439.418,Z 301.637,A -85,B 0,C 180,E1 -9234.847,E2 -9234.847} C_VEL
LIN {X 0,Y 439.188,Z 306.119,A -85,B 0,C 180,E1 -9238.126,E2 -9238.126} C_VEL
LIN {X 0,Y 438.992,Z 310.625,A -85,B 0,C 180,E1 -9241.297,E2 -9241.297} C_VEL
LIN {X 0,Y 438.816,Z 315.139,A -85,B 0,C 180,E1 -9244.379,E2 -9244.379} C_VEL
LIN {X 0,Y 438.711,Z 318.709,A -85,B 0,C 180,E1 -9246.765,E2 -9246.765} C_VEL
LIN {X 0,Y 444.119,Z 337.017,A -85,B 0,C 180,E1 -9247.533,E2 -9247.533} C_VEL
LIN {X 0,Y 447.101,Z 349.611,A -85,B 0,C 180,E1 -9248.158,E2 -9248.158} C_VEL
LIN {X 0,Y 446.272,Z 365.013,A -85,B 0,C 180,E1 -9248.886,E2 -9248.886} C_VEL
LIN {X 0,Y 445.16,Z 379.844,A -85,B 0,C 180,E1 -9249.797,E2 -9249.797} C_VEL
LIN {X 0,Y 444.15,Z 393.234,A -85,B 0,C 180,E1 -9250.833,E2 -9250.833} C_VEL
LIN {X 0,Y 443.108,Z 405.655,A -85,B 0,C 180,E1 -9252.001,E2 -9252.001} C_VEL
LIN {X 0,Y 442.002,Z 417.724,A -85,B 0,C 180,E1 -9253.37,E2 -9253.37} C_VEL
LIN {X 0,Y 441.107,Z 427.945,A -85,B 0,C 180,E1 -9254.759,E2 -9254.759} C_VEL
LIN {X 0,Y 440.246,Z 438.084,A -85,B 0,C 180,E1 -9256.405,E2 -9256.405} C_VEL
LIN {X 0,Y 439.68,Z 446.248,A -85,B 0,C 180,E1 -9258.007,E2 -9258.007} C_VEL
LIN {X 0,Y 439.011,Z 454.046,A -85,B 0,C 180,E1 -9259.858,E2 -9259.858} C_VEL
LIN {X 0,Y 438.843,Z 457.571,A -85,B 0,C 180,E1 -9260.858,E2 -9260.858} C_VEL
LIN {X 0,Y 438.043,Z 459.865,A -85,B 0,C 180,E1 -9261.564,E2 -9261.564} C_VEL
LIN {X 0,Y 435.011,Z 463.245,A -85,B 0,C 180,E1 -9262.722,E2 -9262.722} C_VEL
LIN {X 0,Y 432.49,Z 465.568,A -85,B 0,C 180,E1 -9263.671,E2 -9263.671} C_VEL
LIN {X 0,Y 431.382,Z 467.083,A -85,B 0,C 180,E1 -9264.418,E2 -9264.418} C_VEL
LIN {X 0,Y 431.276,Z 467.518,A -85,B 0,C 180,E1 -9264.673,E2 -9264.673} C_VEL
LIN {X 0,Y 431.174,Z 469.944,A -85,B 0,C 180,E1 -9266.262,E2 -9266.262} C_VEL
LIN {X 0,Y 431.2,Z 471.697,A -85,B 0,C 180,E1 -9268.132,E2 -9268.132} C_VEL
LIN {X 0,Y 431.142,Z 472.31,A -85,B 0,C 180,E1 -9270,E2 -9270} C_VEL
LIN {X 0,Y 431.201,Z 471.746,A -85,B 0,C 180,E1 -9271.868,E2 -9271.868} C_VEL
LIN {X 0,Y 431.174,Z 470.059,A -85,B 0,C 180,E1 -9273.739,E2 -9273.739} C_VEL
LIN {X 0,Y 431.297,Z 467.208,A -85,B 0,C 180,E1 -9275.611,E2 -9275.611} C_VEL
LIN {X 0,Y 431.469,Z 463.127,A -85,B 0,C 180,E1 -9277.488,E2 -9277.488} C_VEL
LIN {X 0,Y 431.758,Z 457.718,A -85,B 0,C 180,E1 -9279.368,E2 -9279.368} C_VEL
LIN {X 0,Y 432.35,Z 450.826,A -85,B 0,C 180,E1 -9281.249,E2 -9281.249} C_VEL
LIN {X 0,Y 432.839,Z 442.748,A -85,B 0,C 180,E1 -9283.038,E2 -9283.038} C_VEL
LIN {X 0,Y 433.755,Z 433.085,A -85,B 0,C 180,E1 -9284.785,E2 -9284.785} C_VEL
LIN {X 0,Y 434.606,Z 423.77,A -85,B 0,C 180,E1 -9286.198,E2 -9286.198} C_VEL
LIN {X 0,Y 435.799,Z 411.335,A -85,B 0,C 180,E1 -9287.767,E2 -9287.767} C_VEL
LIN {X 0,Y 436.896,Z 399.426,A -85,B 0,C 180,E1 -9289.011,E2 -9289.011} C_VEL
LIN {X 0,Y 438.051,Z 385.86,A -85,B 0,C 180,E1 -9290.178,E2 -9290.178} C_VEL
LIN {X 0,Y 439.182,Z 372.519,A -85,B 0,C 180,E1 -9291.104,E2 -9291.104} C_VEL
LIN {X 0,Y 440.076,Z 357.761,A -85,B 0,C 180,E1 -9291.921,E2 -9291.921} C_VEL
LIN {X 0,Y 440.438,Z 350.305,A -85,B 0,C 180,E1 -9292.256,E2 -9292.256} C_VEL
LIN {X 0,Y 436.741,Z 335.835,A -85,B 0,C 180,E1 -9293.005,E2 -9293.005} C_VEL
LIN {X 0,Y 432.346,Z 321.483,A -85,B 0,C 180,E1 -9293.621,E2 -9293.621} C_VEL
LIN {X 0,Y 431.684,Z 318.789,A -85,B 0,C 180,E1 -9293.741,E2 -9293.741} C_VEL
LIN {X 0,Y 431.809,Z 313.895,A -85,B 0,C 180,E1 -9297.111,E2 -9297.111} C_VEL
LIN {X 0,Y 432.064,Z 309.158,A -85,B 0,C 180,E1 -9300.446,E2 -9300.446} C_VEL
LIN {X 0,Y 432.292,Z 304.297,A -85,B 0,C 180,E1 -9303.99,E2 -9303.99} C_VEL
LIN {X 0,Y 432.428,Z 300.365,A -85,B 0,C 180,E1 -9306.966,E2 -9306.966} C_VEL
LIN {X 0,Y 432.667,Z 296.193,A -85,B 0,C 180,E1 -9310.231,E2 -9310.231} C_VEL
LIN {X 0,Y 432.527,Z 292.81,A -85,B 0,C 180,E1 -9313.035,E2 -9313.035} C_VEL
LIN {X 0,Y 432.361,Z 291.306,A -85,B 0,C 180,E1 -9314.343,E2 -9314.343} C_VEL
LIN {X 0,Y 432.319,Z 291.262,A -85,B 0,C 180,E1 -9317.015,E2 -9317.015} C_VEL
LIN {X 0,Y 432.34,Z 291.255,A -85,B 0,C 180,E1 -9319.819,E2 -9319.819} C_VEL
LIN {X 0,Y 432.305,Z 291.264,A -85,B 0,C 180,E1 -9323.022,E2 -9323.022} C_VEL
LIN {X 0,Y 432.357,Z 291.256,A -85,B 0,C 180,E1 -9325.996,E2 -9325.996} C_VEL
LIN {X 0,Y 432.344,Z 291.258,A -85,B 0,C 180,E1 -9329.49,E2 -9329.49} C_VEL
LIN {X 0,Y 432.344,Z 291.255,A -85,B 0,C 180,E1 -9331.874,E2 -9331.874} C_VEL
LIN {X 0,Y 432.376,Z 291.253,A -85,B 0,C 180,E1 -9335.538,E2 -9335.538} C_VEL
LIN {X 0,Y 432.347,Z 291.256,A -85,B 0,C 180,E1 -9339.046,E2 -9339.046} C_VEL
LIN {X 0,Y 432.375,Z 291.253,A -85,B 0,C 180,E1 -9342.011,E2 -9342.011} C_VEL
LIN {X 0,Y 432.39,Z 291.252,A -85,B 0,C 180,E1 -9344.926,E2 -9344.926} C_VEL
LIN {X 0,Y 432.456,Z 291.242,A -85,B 0,C 180,E1 -9347.803,E2 -9347.803} C_VEL
LIN {X 0,Y 432.461,Z 291.239,A -85,B 0,C 180,E1 -9351.59,E2 -9351.59} C_VEL
LIN {X 0,Y 432.579,Z 291.226,A -85,B 0,C 180,E1 -9354.406,E2 -9354.406} C_VEL
LIN {X 0,Y 432.603,Z 291.223,A -85,B 0,C 180,E1 -9358.138,E2 -9358.138} C_VEL
LIN {X 0,Y 432.723,Z 291.211,A -85,B 0,C 180,E1 -9360,E2 -9360} C_VEL
LIN {X 0,Y 432.603,Z 291.224,A -85,B 0,C 180,E1 -9362.793,E2 -9362.793} C_VEL
LIN {X 0,Y 432.579,Z 291.225,A -85,B 0,C 180,E1 -9365.594,E2 -9365.594} C_VEL
LIN {X 0,Y 432.461,Z 291.24,A -85,B 0,C 180,E1 -9368.41,E2 -9368.41} C_VEL
LIN {X 0,Y 432.456,Z 291.245,A -85,B 0,C 180,E1 -9372.197,E2 -9372.197} C_VEL
LIN {X 0,Y 432.427,Z 291.244,A -85,B 0,C 180,E1 -9376.039,E2 -9376.039} C_VEL
LIN {X 0,Y 432.384,Z 291.251,A -85,B 0,C 180,E1 -9379.485,E2 -9379.485} C_VEL
LIN {X 0,Y 432.315,Z 291.262,A -85,B 0,C 180,E1 -9382.964,E2 -9382.964} C_VEL
LIN {X 0,Y 432.359,Z 291.257,A -85,B 0,C 180,E1 -9386.033,E2 -9386.033} C_VEL
LIN {X 0,Y 432.339,Z 291.261,A -85,B 0,C 180,E1 -9389.188,E2 -9389.188} C_VEL
LIN {X 0,Y 432.32,Z 291.264,A -85,B 0,C 180,E1 -9392.443,E2 -9392.443} C_VEL
LIN {X 0,Y 432.341,Z 291.262,A -85,B 0,C 180,E1 -9395.632,E2 -9395.632} C_VEL
LIN {X 0,Y 432.331,Z 291.261,A -85,B 0,C 180,E1 -9398.713,E2 -9398.713} C_VEL
LIN {X 0,Y 432.322,Z 291.26,A -85,B 0,C 180,E1 -9401.798,E2 -9401.798} C_VEL
LIN {X 0,Y 432.313,Z 291.264,A -85,B 0,C 180,E1 -9403.061,E2 -9403.061} C_VEL
LIN {X 0,Y 432.468,Z 291.975,A -85,B 0,C 180,E1 -9404.354,E2 -9404.354} C_VEL
LIN {X 0,Y 432.952,Z 295.482,A -85,B 0,C 180,E1 -9407.018,E2 -9407.018} C_VEL
LIN {X 0,Y 433.053,Z 298.987,A -85,B 0,C 180,E1 -9409.522,E2 -9409.522} C_VEL
LIN {X 0,Y 432.826,Z 303.706,A -85,B 0,C 180,E1 -9412.715,E2 -9412.715} C_VEL
LIN {X 0,Y 432.556,Z 308.719,A -85,B 0,C 180,E1 -9415.958,E2 -9415.958} C_VEL
LIN {X 0,Y 432.227,Z 314.8,A -85,B 0,C 180,E1 -9419.731,E2 -9419.731} C_VEL
LIN {X 0,Y 431.896,Z 320.097,A -85,B 0,C 180,E1 -9422.895,E2 -9422.895} C_VEL
LIN {X 0,Y 431.726,Z 325.978,A -85,B 0,C 180,E1 -9426.324,E2 -9426.324} C_VEL
LIN {X 0,Y 434.05,Z 334.112,A -85,B 0,C 180,E1 -9426.625,E2 -9426.625} C_VEL
LIN {X 0,Y 438.339,Z 349.956,A -85,B 0,C 180,E1 -9427.342,E2 -9427.342} C_VEL
LIN {X 0,Y 440.223,Z 358.968,A -85,B 0,C 180,E1 -9427.812,E2 -9427.812} C_VEL
LIN {X 0,Y 439.449,Z 373.831,A -85,B 0,C 180,E1 -9428.541,E2 -9428.541} C_VEL
LIN {X 0,Y 438.436,Z 386.908,A -85,B 0,C 180,E1 -9429.35,E2 -9429.35} C_VEL
LIN {X 0,Y 437.322,Z 400.495,A -85,B 0,C 180,E1 -9430.399,E2 -9430.399} C_VEL
LIN {X 0,Y 436.095,Z 414.052,A -85,B 0,C 180,E1 -9431.684,E2 -9431.684} C_VEL
LIN {X 0,Y 434.977,Z 426.243,A -85,B 0,C 180,E1 -9433.092,E2 -9433.092} C_VEL
LIN {X 0,Y 434.001,Z 436.471,A -85,B 0,C 180,E1 -9434.503,E2 -9434.503} C_VEL
LIN {X 0,Y 433.109,Z 446.467,A -85,B 0,C 180,E1 -9436.152,E2 -9436.152} C_VEL
LIN {X 0,Y 432.417,Z 454.766,A -85,B 0,C 180,E1 -9437.802,E2 -9437.802} C_VEL
LIN {X 0,Y 432.025,Z 460.75,A -85,B 0,C 180,E1 -9439.218,E2 -9439.218} C_VEL
LIN {X 0,Y 431.599,Z 467.336,A -85,B 0,C 180,E1 -9441.101,E2 -9441.101} C_VEL
LIN {X 0,Y 431.379,Z 472.489,A -85,B 0,C 180,E1 -9442.981,E2 -9442.981} C_VEL
LIN {X 0,Y 431.251,Z 475.469,A -85,B 0,C 180,E1 -9444.388,E2 -9444.388} C_VEL
LIN {X 0,Y 431.146,Z 478.371,A -85,B 0,C 180,E1 -9446.261,E2 -9446.261} C_VEL
LIN {X 0,Y 431.193,Z 480.104,A -85,B 0,C 180,E1 -9448.132,E2 -9448.132} C_VEL
LIN {X 0,Y 431.141,Z 480.697,A -85,B 0,C 180,E1 -9450,E2 -9450} C_VEL
LIN {X 0,Y 431.193,Z 480.101,A -85,B 0,C 180,E1 -9451.868,E2 -9451.868} C_VEL
LIN {X 0,Y 431.146,Z 478.365,A -85,B 0,C 180,E1 -9453.738,E2 -9453.738} C_VEL
LIN {X 0,Y 431.266,Z 475.464,A -85,B 0,C 180,E1 -9455.611,E2 -9455.611} C_VEL
LIN {X 0,Y 431.409,Z 471.327,A -85,B 0,C 180,E1 -9457.488,E2 -9457.488} C_VEL
LIN {X 0,Y 431.671,Z 465.844,A -85,B 0,C 180,E1 -9459.369,E2 -9459.369} C_VEL
LIN {X 0,Y 432.197,Z 458.866,A -85,B 0,C 180,E1 -9461.252,E2 -9461.252} C_VEL
LIN {X 0,Y 432.8,Z 450.178,A -85,B 0,C 180,E1 -9463.14,E2 -9463.14} C_VEL
LIN {X 0,Y 433.619,Z 440.949,A -85,B 0,C 180,E1 -9464.789,E2 -9464.789} C_VEL
LIN {X 0,Y 434.47,Z 431.562,A -85,B 0,C 180,E1 -9466.202,E2 -9466.202} C_VEL
LIN {X 0,Y 435.571,Z 419.8,A -85,B 0,C 180,E1 -9467.683,E2 -9467.683} C_VEL
LIN {X 0,Y 436.729,Z 406.975,A -85,B 0,C 180,E1 -9469.018,E2 -9469.018} C_VEL
LIN {X 0,Y 437.897,Z 393.236,A -85,B 0,C 180,E1 -9470.185,E2 -9470.185} C_VEL
LIN {X 0,Y 439.025,Z 379.742,A -85,B 0,C 180,E1 -9471.111,E2 -9471.111} C_VEL
LIN {X 0,Y 439.919,Z 365.9,A -85,B 0,C 180,E1 -9471.87,E2 -9471.87} C_VEL
LIN {X 0,Y 440.196,Z 359.114,A -85,B 0,C 180,E1 -9472.18,E2 -9472.18} C_VEL
LIN {X 0,Y 437.109,Z 345.212,A -85,B 0,C 180,E1 -9472.883,E2 -9472.883} C_VEL
LIN {X 0,Y 432.66,Z 329.639,A -85,B 0,C 180,E1 -9473.543,E2 -9473.543} C_VEL
LIN {X 0,Y 431.715,Z 325.985,A -85,B 0,C 180,E1 -9473.68,E2 -9473.68} C_VEL
LIN {X 0,Y 431.895,Z 320.133,A -85,B 0,C 180,E1 -9477.105,E2 -9477.105} C_VEL
LIN {X 0,Y 432.24,Z 314.513,A -85,B 0,C 180,E1 -9480.486,E2 -9480.486} C_VEL
LIN {X 0,Y 432.554,Z 308.766,A -85,B 0,C 180,E1 -9484.042,E2 -9484.042} C_VEL
LIN {X 0,Y 432.823,Z 303.723,A -85,B 0,C 180,E1 -9487.284,E2 -9487.284} C_VEL
LIN {X 0,Y 433.048,Z 298.977,A -85,B 0,C 180,E1 -9490.478,E2 -9490.478} C_VEL
LIN {X 0,Y 432.948,Z 295.463,A -85,B 0,C 180,E1 -9492.982,E2 -9492.982} C_VEL
LIN {X 0,Y 432.465,Z 291.919,A -85,B 0,C 180,E1 -9495.67,E2 -9495.67} C_VEL
LIN {X 0,Y 432.317,Z 291.263,A -85,B 0,C 180,E1 -9497.015,E2 -9497.015} C_VEL
LIN {X 0,Y 432.33,Z 291.26,A -85,B 0,C 180,E1 -9499.82,E2 -9499.82} C_VEL
LIN {X 0,Y 432.299,Z 291.265,A -85,B 0,C 180,E1 -9503.021,E2 -9503.021} C_VEL
LIN {X 0,Y 432.352,Z 291.259,A -85,B 0,C 180,E1 -9505.996,E2 -9505.996} C_VEL
LIN {X 0,Y 432.34,Z 291.262,A -85,B 0,C 180,E1 -9509.489,E2 -9509.489} C_VEL
LIN {X 0,Y 432.383,Z 291.252,A -85,B 0,C 180,E1 -9512.928,E2 -9512.928} C_VEL
LIN {X 0,Y 432.363,Z 291.253,A -85,B 0,C 180,E1 -9516.023,E2 -9516.023} C_VEL
LIN {X 0,Y 432.342,Z 291.256,A -85,B 0,C 180,E1 -9519.046,E2 -9519.046} C_VEL
LIN {X 0,Y 432.37,Z 291.252,A -85,B 0,C 180,E1 -9522.011,E2 -9522.011} C_VEL
LIN {X 0,Y 432.386,Z 291.25,A -85,B 0,C 180,E1 -9524.926,E2 -9524.926} C_VEL
LIN {X 0,Y 432.452,Z 291.243,A -85,B 0,C 180,E1 -9527.803,E2 -9527.803} C_VEL
LIN {X 0,Y 432.456,Z 291.24,A -85,B 0,C 180,E1 -9531.59,E2 -9531.59} C_VEL
LIN {X 0,Y 432.575,Z 291.224,A -85,B 0,C 180,E1 -9534.406,E2 -9534.406} C_VEL
LIN {X 0,Y 432.597,Z 291.221,A -85,B 0,C 180,E1 -9538.138,E2 -9538.138} C_VEL
LIN {X 0,Y 432.721,Z 291.211,A -85,B 0,C 180,E1 -9540,E2 -9540} C_VEL
LIN {X 0,Y 432.599,Z 291.224,A -85,B 0,C 180,E1 -9542.794,E2 -9542.794} C_VEL
LIN {X 0,Y 432.515,Z 291.234,A -85,B 0,C 180,E1 -9546.46,E2 -9546.46} C_VEL
LIN {X 0,Y 432.433,Z 291.247,A -85,B 0,C 180,E1 -9549.353,E2 -9549.353} C_VEL
LIN {X 0,Y 432.423,Z 291.245,A -85,B 0,C 180,E1 -9552.804,E2 -9552.804} C_VEL
LIN {X 0,Y 432.405,Z 291.249,A -85,B 0,C 180,E1 -9556.479,E2 -9556.479} C_VEL
LIN {X 0,Y 432.331,Z 291.258,A -85,B 0,C 180,E1 -9559.961,E2 -9559.961} C_VEL
LIN {X 0,Y 432.312,Z 291.263,A -85,B 0,C 180,E1 -9562.965,E2 -9562.965} C_VEL
LIN {X 0,Y 432.357,Z 291.256,A -85,B 0,C 180,E1 -9566.033,E2 -9566.033} C_VEL
LIN {X 0,Y 432.336,Z 291.257,A -85,B 0,C 180,E1 -9569.188,E2 -9569.188} C_VEL
LIN {X 0,Y 432.317,Z 291.257,A -85,B 0,C 180,E1 -9572.444,E2 -9572.444} C_VEL
LIN {X 0,Y 432.338,Z 291.255,A -85,B 0,C 180,E1 -9575.632,E2 -9575.632} C_VEL
LIN {X 0,Y 432.349,Z 291.256,A -85,B 0,C 180,E1 -9579.343,E2 -9579.343} C_VEL
LIN {X 0,Y 432.328,Z 291.259,A -85,B 0,C 180,E1 -9581.798,E2 -9581.798} C_VEL
LIN {X 0,Y 432.329,Z 291.26,A -85,B 0,C 180,E1 -9584.348,E2 -9584.348} C_VEL
LIN {X 0,Y 432.331,Z 291.26,A -85,B 0,C 180,E1 -9585.665,E2 -9585.665} C_VEL
LIN {X 0,Y 432.61,Z 294.335,A -85,B 0,C 180,E1 -9588.357,E2 -9588.357} C_VEL
LIN {X 0,Y 432.584,Z 297.198,A -85,B 0,C 180,E1 -9590.684,E2 -9590.684} C_VEL
LIN {X 0,Y 432.39,Z 301.916,A -85,B 0,C 180,E1 -9594.36,E2 -9594.36} C_VEL
LIN {X 0,Y 432.16,Z 306.443,A -85,B 0,C 180,E1 -9597.742,E2 -9597.742} C_VEL
LIN {X 0,Y 431.961,Z 310.686,A -85,B 0,C 180,E1 -9600.785,E2 -9600.785} C_VEL
LIN {X 0,Y 431.794,Z 315.206,A -85,B 0,C 180,E1 -9603.931,E2 -9603.931} C_VEL
LIN {X 0,Y 431.66,Z 318.806,A -85,B 0,C 180,E1 -9606.38,E2 -9606.38} C_VEL
LIN {X 0,Y 436.175,Z 333.699,A -85,B 0,C 180,E1 -9606.992,E2 -9606.992} C_VEL
LIN {X 0,Y 440.063,Z 348.693,A -85,B 0,C 180,E1 -9607.75,E2 -9607.75} C_VEL
LIN {X 0,Y 440.369,Z 352.399,A -85,B 0,C 180,E1 -9607.932,E2 -9607.932} C_VEL
LIN {X 0,Y 439.491,Z 367.084,A -85,B 0,C 180,E1 -9608.667,E2 -9608.667} C_VEL
LIN {X 0,Y 438.503,Z 379.919,A -85,B 0,C 180,E1 -9609.477,E2 -9609.477} C_VEL
LIN {X 0,Y 437.417,Z 393.309,A -85,B 0,C 180,E1 -9610.526,E2 -9610.526} C_VEL
LIN {X 0,Y 436.365,Z 405.579,A -85,B 0,C 180,E1 -9611.697,E2 -9611.697} C_VEL
LIN {X 0,Y 435.167,Z 417.797,A -85,B 0,C 180,E1 -9613.101,E2 -9613.101} C_VEL
LIN {X 0,Y 434.227,Z 428.018,A -85,B 0,C 180,E1 -9614.512,E2 -9614.512} C_VEL
LIN {X 0,Y 433.303,Z 438.022,A -85,B 0,C 180,E1 -9616.159,E2 -9616.159} C_VEL
LIN {X 0,Y 432.66,Z 446.32,A -85,B 0,C 180,E1 -9617.81,E2 -9617.81} C_VEL
LIN {X 0,Y 432.138,Z 452.313,A -85,B 0,C 180,E1 -9619.221,E2 -9619.221} C_VEL
LIN {X 0,Y 431.714,Z 458.905,A -85,B 0,C 180,E1 -9621.104,E2 -9621.104} C_VEL
LIN {X 0,Y 431.407,Z 464.061,A -85,B 0,C 180,E1 -9622.982,E2 -9622.982} C_VEL
LIN {X 0,Y 431.276,Z 467.518,A -85,B 0,C 180,E1 -9624.673,E2 -9624.673} C_VEL
LIN {X 0,Y 430.558,Z 468.835,A -85,B 0,C 180,E1 -9625.435,E2 -9625.435} C_VEL
LIN {X 0,Y 427.654,Z 470.513,A -85,B 0,C 180,E1 -9626.681,E2 -9626.681} C_VEL
LIN {X 0,Y 425.218,Z 471.472,A -85,B 0,C 180,E1 -9627.694,E2 -9627.694} C_VEL
LIN {X 0,Y 424.165,Z 471.957,A -85,B 0,C 180,E1 -9628.481,E2 -9628.481} C_VEL
LIN {X 0,Y 424.073,Z 472.076,A -85,B 0,C 180,E1 -9628.748,E2 -9628.748} C_VEL
LIN {X 0,Y 424.06,Z 472.379,A -85,B 0,C 180,E1 -9630,E2 -9630} C_VEL
LIN {X 0,Y 424.127,Z 471.815,A -85,B 0,C 180,E1 -9631.9,E2 -9631.9} C_VEL
LIN {X 0,Y 424.084,Z 470.127,A -85,B 0,C 180,E1 -9633.801,E2 -9633.801} C_VEL
LIN {X 0,Y 424.21,Z 467.276,A -85,B 0,C 180,E1 -9635.705,E2 -9635.705} C_VEL
LIN {X 0,Y 424.391,Z 463.196,A -85,B 0,C 180,E1 -9637.613,E2 -9637.613} C_VEL
LIN {X 0,Y 424.707,Z 457.786,A -85,B 0,C 180,E1 -9639.525,E2 -9639.525} C_VEL
LIN {X 0,Y 425.355,Z 450.893,A -85,B 0,C 180,E1 -9641.436,E2 -9641.436} C_VEL
LIN {X 0,Y 425.957,Z 442.293,A -85,B 0,C 180,E1 -9643.356,E2 -9643.356} C_VEL
LIN {X 0,Y 426.842,Z 433.151,A -85,B 0,C 180,E1 -9645.03,E2 -9645.03} C_VEL
LIN {X 0,Y 427.757,Z 423.836,A -85,B 0,C 180,E1 -9646.464,E2 -9646.464} C_VEL
LIN {X 0,Y 428.947,Z 412.027,A -85,B 0,C 180,E1 -9647.986,E2 -9647.986} C_VEL
LIN {X 0,Y 430.135,Z 399.491,A -85,B 0,C 180,E1 -9649.321,E2 -9649.321} C_VEL
LIN {X 0,Y 431.347,Z 385.923,A -85,B 0,C 180,E1 -9650.506,E2 -9650.506} C_VEL
LIN {X 0,Y 432.56,Z 372.581,A -85,B 0,C 180,E1 -9651.443,E2 -9651.443} C_VEL
LIN {X 0,Y 433.473,Z 357.822,A -85,B 0,C 180,E1 -9652.272,E2 -9652.272} C_VEL
LIN {X 0,Y 433.768,Z 351.715,A -85,B 0,C 180,E1 -9652.553,E2 -9652.553} C_VEL
LIN {X 0,Y 430.137,Z 337.246,A -85,B 0,C 180,E1 -9653.332,E2 -9653.332} C_VEL
LIN {X 0,Y 425.551,Z 322.13,A -85,B 0,C 180,E1 -9654.009,E2 -9654.009} C_VEL
LIN {X 0,Y 424.628,Z 318.889,A -85,B 0,C 180,E1 -9654.138,E2 -9654.138} C_VEL
LIN {X 0,Y 424.791,Z 313.958,A -85,B 0,C 180,E1 -9657.597,E2 -9657.597} C_VEL
LIN {X 0,Y 425.012,Z 309.462,A -85,B 0,C 180,E1 -9660.838,E2 -9660.838} C_VEL
LIN {X 0,Y 425.268,Z 304.82,A -85,B 0,C 180,E1 -9664.279,E2 -9664.279} C_VEL
LIN {X 0,Y 425.426,Z 300.422,A -85,B 0,C 180,E1 -9667.679,E2 -9667.679} C_VEL
LIN {X 0,Y 425.639,Z 296.795,A -85,B 0,C 180,E1 -9670.577,E2 -9670.577} C_VEL
LIN {X 0,Y 425.473,Z 293.482,A -85,B 0,C 180,E1 -9673.381,E2 -9673.381} C_VEL
LIN {X 0,Y 425.302,Z 292.137,A -85,B 0,C 180,E1 -9674.719,E2 -9674.719} C_VEL
LIN {X 0,Y 425.289,Z 292.135,A -85,B 0,C 180,E1 -9678.042,E2 -9678.042} C_VEL
LIN {X 0,Y 425.311,Z 292.132,A -85,B 0,C 180,E1 -9681.103,E2 -9681.103} C_VEL
LIN {X 0,Y 425.297,Z 292.137,A -85,B 0,C 180,E1 -9684.664,E2 -9684.664} C_VEL
LIN {X 0,Y 425.263,Z 292.141,A -85,B 0,C 180,E1 -9688.073,E2 -9688.073} C_VEL
LIN {X 0,Y 425.311,Z 292.132,A -85,B 0,C 180,E1 -9691.366,E2 -9691.366} C_VEL
LIN {X 0,Y 425.27,Z 292.137,A -85,B 0,C 180,E1 -9694.553,E2 -9694.553} C_VEL
LIN {X 0,Y 425.282,Z 292.135,A -85,B 0,C 180,E1 -9696.633,E2 -9696.633} C_VEL
LIN {X 0,Y 425.293,Z 292.134,A -85,B 0,C 180,E1 -9699.694,E2 -9699.694} C_VEL
LIN {X 0,Y 425.339,Z 292.128,A -85,B 0,C 180,E1 -9702.697,E2 -9702.697} C_VEL
LIN {X 0,Y 425.343,Z 292.127,A -85,B 0,C 180,E1 -9705.65,E2 -9705.65} C_VEL
LIN {X 0,Y 425.349,Z 292.126,A -85,B 0,C 180,E1 -9708.564,E2 -9708.564} C_VEL
LIN {X 0,Y 425.405,Z 292.118,A -85,B 0,C 180,E1 -9711.449,E2 -9711.449} C_VEL
LIN {X 0,Y 425.532,Z 292.105,A -85,B 0,C 180,E1 -9714.313,E2 -9714.313} C_VEL
LIN {X 0,Y 425.572,Z 292.099,A -85,B 0,C 180,E1 -9718.107,E2 -9718.107} C_VEL
LIN {X 0,Y 425.693,Z 292.086,A -85,B 0,C 180,E1 -9720,E2 -9720} C_VEL
LIN {X 0,Y 425.554,Z 292.103,A -85,B 0,C 180,E1 -9722.84,E2 -9722.84} C_VEL
LIN {X 0,Y 425.532,Z 292.104,A -85,B 0,C 180,E1 -9725.687,E2 -9725.687} C_VEL
LIN {X 0,Y 425.405,Z 292.119,A -85,B 0,C 180,E1 -9728.551,E2 -9728.551} C_VEL
LIN {X 0,Y 425.409,Z 292.122,A -85,B 0,C 180,E1 -9732.402,E2 -9732.402} C_VEL
LIN {X 0,Y 425.385,Z 292.122,A -85,B 0,C 180,E1 -9736.312,E2 -9736.312} C_VEL
LIN {X 0,Y 425.325,Z 292.131,A -85,B 0,C 180,E1 -9739.636,E2 -9739.636} C_VEL
LIN {X 0,Y 425.285,Z 292.134,A -85,B 0,C 180,E1 -9742.339,E2 -9742.339} C_VEL
LIN {X 0,Y 425.29,Z 292.133,A -85,B 0,C 180,E1 -9745.446,E2 -9745.446} C_VEL
LIN {X 0,Y 425.328,Z 292.132,A -85,B 0,C 180,E1 -9748.632,E2 -9748.632} C_VEL
LIN {X 0,Y 425.262,Z 292.143,A -85,B 0,C 180,E1 -9751.927,E2 -9751.927} C_VEL
LIN {X 0,Y 425.296,Z 292.142,A -85,B 0,C 180,E1 -9755.336,E2 -9755.336} C_VEL
LIN {X 0,Y 425.29,Z 292.138,A -85,B 0,C 180,E1 -9758.899,E2 -9758.899} C_VEL
LIN {X 0,Y 425.28,Z 292.137,A -85,B 0,C 180,E1 -9761.957,E2 -9761.957} C_VEL
LIN {X 0,Y 425.282,Z 292.14,A -85,B 0,C 180,E1 -9763.355,E2 -9763.355} C_VEL
LIN {X 0,Y 425.794,Z 295.443,A -85,B 0,C 180,E1 -9766.113,E2 -9766.113} C_VEL
LIN {X 0,Y 426.05,Z 298.94,A -85,B 0,C 180,E1 -9768.714,E2 -9768.714} C_VEL
LIN {X 0,Y 425.934,Z 302.442,A -85,B 0,C 180,E1 -9771.171,E2 -9771.171} C_VEL
LIN {X 0,Y 425.61,Z 307.703,A -85,B 0,C 180,E1 -9774.694,E2 -9774.694} C_VEL
LIN {X 0,Y 425.337,Z 311.956,A -85,B 0,C 180,E1 -9777.425,E2 -9777.425} C_VEL
LIN {X 0,Y 425.087,Z 316.502,A -85,B 0,C 180,E1 -9780.265,E2 -9780.265} C_VEL
LIN {X 0,Y 424.803,Z 321.795,A -85,B 0,C 180,E1 -9783.468,E2 -9783.468} C_VEL
LIN {X 0,Y 424.679,Z 325.911,A -85,B 0,C 180,E1 -9785.907,E2 -9785.907} C_VEL
LIN {X 0,Y 428.434,Z 338.851,A -85,B 0,C 180,E1 -9786.429,E2 -9786.429} C_VEL
LIN {X 0,Y 432.083,Z 353.222,A -85,B 0,C 180,E1 -9787.13,E2 -9787.13} C_VEL
LIN {X 0,Y 433.587,Z 360.987,A -85,B 0,C 180,E1 -9787.554,E2 -9787.554} C_VEL
LIN {X 0,Y 432.653,Z 375.756,A -85,B 0,C 180,E1 -9788.312,E2 -9788.312} C_VEL
LIN {X 0,Y 431.505,Z 390.045,A -85,B 0,C 180,E1 -9789.253,E2 -9789.253} C_VEL
LIN {X 0,Y 430.331,Z 403.051,A -85,B 0,C 180,E1 -9790.316,E2 -9790.316} C_VEL
LIN {X 0,Y 429.096,Z 416.128,A -85,B 0,C 180,E1 -9791.622,E2 -9791.622} C_VEL
LIN {X 0,Y 427.943,Z 427.961,A -85,B 0,C 180,E1 -9793.052,E2 -9793.052} C_VEL
LIN {X 0,Y 426.951,Z 437.917,A -85,B 0,C 180,E1 -9794.485,E2 -9794.485} C_VEL
LIN {X 0,Y 426.034,Z 447.655,A -85,B 0,C 180,E1 -9796.161,E2 -9796.161} C_VEL
LIN {X 0,Y 425.36,Z 455.78,A -85,B 0,C 180,E1 -9797.839,E2 -9797.839} C_VEL
LIN {X 0,Y 424.808,Z 462.493,A -85,B 0,C 180,E1 -9799.515,E2 -9799.515} C_VEL
LIN {X 0,Y 424.475,Z 468.694,A -85,B 0,C 180,E1 -9801.43,E2 -9801.43} C_VEL
LIN {X 0,Y 424.243,Z 473.489,A -85,B 0,C 180,E1 -9803.341,E2 -9803.341} C_VEL
LIN {X 0,Y 424.151,Z 477.002,A -85,B 0,C 180,E1 -9805.247,E2 -9805.247} C_VEL
LIN {X 0,Y 424.076,Z 479.312,A -85,B 0,C 180,E1 -9807.15,E2 -9807.15} C_VEL
LIN {X 0,Y 424.066,Z 480.475,A -85,B 0,C 180,E1 -9809.05,E2 -9809.05} C_VEL
LIN {X 0,Y 424.066,Z 480.473,A -85,B 0,C 180,E1 -9810.949,E2 -9810.949} C_VEL
LIN {X 0,Y 424.076,Z 479.306,A -85,B 0,C 180,E1 -9812.849,E2 -9812.849} C_VEL
LIN {X 0,Y 424.154,Z 476.994,A -85,B 0,C 180,E1 -9814.752,E2 -9814.752} C_VEL
LIN {X 0,Y 424.293,Z 473.487,A -85,B 0,C 180,E1 -9816.658,E2 -9816.658} C_VEL
LIN {X 0,Y 424.474,Z 468.692,A -85,B 0,C 180,E1 -9818.569,E2 -9818.569} C_VEL
LIN {X 0,Y 424.807,Z 462.482,A -85,B 0,C 180,E1 -9820.485,E2 -9820.485} C_VEL
LIN {X 0,Y 425.362,Z 455.764,A -85,B 0,C 180,E1 -9822.16,E2 -9822.16} C_VEL
LIN {X 0,Y 426.029,Z 447.641,A -85,B 0,C 180,E1 -9823.839,E2 -9823.839} C_VEL
LIN {X 0,Y 426.94,Z 437.9,A -85,B 0,C 180,E1 -9825.515,E2 -9825.515} C_VEL
LIN {X 0,Y 427.968,Z 427.94,A -85,B 0,C 180,E1 -9826.946,E2 -9826.946} C_VEL
LIN {X 0,Y 429.093,Z 416.108,A -85,B 0,C 180,E1 -9828.378,E2 -9828.378} C_VEL
LIN {X 0,Y 430.203,Z 404.315,A -85,B 0,C 180,E1 -9829.566,E2 -9829.566} C_VEL
LIN {X 0,Y 431.351,Z 391.578,A -85,B 0,C 180,E1 -9830.63,E2 -9830.63} C_VEL
LIN {X 0,Y 432.527,Z 377.681,A -85,B 0,C 180,E1 -9831.569,E2 -9831.569} C_VEL
LIN {X 0,Y 433.482,Z 363.132,A -85,B 0,C 180,E1 -9832.344,E2 -9832.344} C_VEL
LIN {X 0,Y 433.303,Z 358.934,A -85,B 0,C 180,E1 -9832.557,E2 -9832.557} C_VEL
LIN {X 0,Y 430.211,Z 345.456,A -85,B 0,C 180,E1 -9833.26,E2 -9833.26} C_VEL
LIN {X 0,Y 425.788,Z 330.064,A -85,B 0,C 180,E1 -9833.936,E2 -9833.936} C_VEL
LIN {X 0,Y 424.686,Z 325.893,A -85,B 0,C 180,E1 -9834.11,E2 -9834.11} C_VEL
LIN {X 0,Y 424.883,Z 320.069,A -85,B 0,C 180,E1 -9837.59,E2 -9837.59} C_VEL
LIN {X 0,Y 425.21,Z 314.807,A -85,B 0,C 180,E1 -9840.821,E2 -9840.821} C_VEL
LIN {X 0,Y 425.539,Z 309.249,A -85,B 0,C 180,E1 -9844.333,E2 -9844.333} C_VEL
LIN {X 0,Y 425.825,Z 304.211,A -85,B 0,C 180,E1 -9847.636,E2 -9847.636} C_VEL
LIN {X 0,Y 426.026,Z 299.848,A -85,B 0,C 180,E1 -9850.638,E2 -9850.638} C_VEL
LIN {X 0,Y 425.97,Z 297.176,A -85,B 0,C 180,E1 -9852.566,E2 -9852.566} C_VEL
LIN {X 0,Y 425.549,Z 293.663,A -85,B 0,C 180,E1 -9855.246,E2 -9855.246} C_VEL
LIN {X 0,Y 425.282,Z 292.139,A -85,B 0,C 180,E1 -9856.644,E2 -9856.644} C_VEL
LIN {X 0,Y 425.284,Z 292.138,A -85,B 0,C 180,E1 -9859.873,E2 -9859.873} C_VEL
LIN {X 0,Y 425.271,Z 292.138,A -85,B 0,C 180,E1 -9862.488,E2 -9862.488} C_VEL
LIN {X 0,Y 425.3,Z 292.137,A -85,B 0,C 180,E1 -9865.817,E2 -9865.817} C_VEL
LIN {X 0,Y 425.283,Z 292.141,A -85,B 0,C 180,E1 -9869.238,E2 -9869.238} C_VEL
LIN {X 0,Y 425.341,Z 292.132,A -85,B 0,C 180,E1 -9872.442,E2 -9872.442} C_VEL
LIN {X 0,Y 425.344,Z 292.13,A -85,B 0,C 180,E1 -9875.602,E2 -9875.602} C_VEL
LIN {X 0,Y 425.285,Z 292.137,A -85,B 0,C 180,E1 -9878.681,E2 -9878.681} C_VEL
LIN {X 0,Y 425.325,Z 292.132,A -85,B 0,C 180,E1 -9881.702,E2 -9881.702} C_VEL
LIN {X 0,Y 425.339,Z 292.129,A -85,B 0,C 180,E1 -9884.67,E2 -9884.67} C_VEL
LIN {X 0,Y 425.404,Z 292.121,A -85,B 0,C 180,E1 -9887.598,E2 -9887.598} C_VEL
LIN {X 0,Y 425.4,Z 292.118,A -85,B 0,C 180,E1 -9891.449,E2 -9891.449} C_VEL
LIN {X 0,Y 425.528,Z 292.102,A -85,B 0,C 180,E1 -9894.313,E2 -9894.313} C_VEL
LIN {X 0,Y 425.567,Z 292.097,A -85,B 0,C 180,E1 -9898.107,E2 -9898.107} C_VEL
LIN {X 0,Y 425.69,Z 292.087,A -85,B 0,C 180,E1 -9900,E2 -9900} C_VEL
LIN {X 0,Y 425.551,Z 292.103,A -85,B 0,C 180,E1 -9902.84,E2 -9902.84} C_VEL
LIN {X 0,Y 425.475,Z 292.11,A -85,B 0,C 180,E1 -9906.458,E2 -9906.458} C_VEL
LIN {X 0,Y 425.392,Z 292.122,A -85,B 0,C 180,E1 -9909.51,E2 -9909.51} C_VEL
LIN {X 0,Y 425.385,Z 292.122,A -85,B 0,C 180,E1 -9912.904,E2 -9912.904} C_VEL
LIN {X 0,Y 425.354,Z 292.128,A -85,B 0,C 180,E1 -9916.605,E2 -9916.605} C_VEL
LIN {X 0,Y 425.321,Z 292.132,A -85,B 0,C 180,E1 -9919.636,E2 -9919.636} C_VEL
LIN {X 0,Y 425.3,Z 292.133,A -85,B 0,C 180,E1 -9923.366,E2 -9923.366} C_VEL
LIN {X 0,Y 425.34,Z 292.126,A -85,B 0,C 180,E1 -9926.845,E2 -9926.845} C_VEL
LIN {X 0,Y 425.284,Z 292.132,A -85,B 0,C 180,E1 -9929.72,E2 -9929.72} C_VEL
LIN {X 0,Y 425.276,Z 292.133,A -85,B 0,C 180,E1 -9933.049,E2 -9933.049} C_VEL
LIN {X 0,Y 425.276,Z 292.134,A -85,B 0,C 180,E1 -9935.929,E2 -9935.929} C_VEL
LIN {X 0,Y 425.295,Z 292.134,A -85,B 0,C 180,E1 -9939.045,E2 -9939.045} C_VEL
LIN {X 0,Y 425.27,Z 292.14,A -85,B 0,C 180,E1 -9942.654,E2 -9942.654} C_VEL
LIN {X 0,Y 425.282,Z 292.136,A -85,B 0,C 180,E1 -9945.284,E2 -9945.284} C_VEL
LIN {X 0,Y 425.512,Z 294.235,A -85,B 0,C 180,E1 -9947.378,E2 -9947.378} C_VEL
LIN {X 0,Y 425.63,Z 297.24,A -85,B 0,C 180,E1 -9949.913,E2 -9949.913} C_VEL
LIN {X 0,Y 425.371,Z 301.748,A -85,B 0,C 180,E1 -9953.503,E2 -9953.503} C_VEL
LIN {X 0,Y 425.25,Z 304.739,A -85,B 0,C 180,E1 -9955.813,E2 -9955.813} C_VEL
LIN {X 0,Y 425.007,Z 309.432,A -85,B 0,C 180,E1 -9959.303,E2 -9959.303} C_VEL
LIN {X 0,Y 424.795,Z 313.767,A -85,B 0,C 180,E1 -9962.404,E2 -9962.404} C_VEL
LIN {X 0,Y 424.63,Z 318.863,A -85,B 0,C 180,E1 -9965.956,E2 -9965.956} C_VEL
LIN {X 0,Y 427.833,Z 329.404,A -85,B 0,C 180,E1 -9966.393,E2 -9966.393} C_VEL
LIN {X 0,Y 431.848,Z 343.638,A -85,B 0,C 180,E1 -9967.089,E2 -9967.089} C_VEL
LIN {X 0,Y 433.755,Z 351.907,A -85,B 0,C 180,E1 -9967.55,E2 -9967.55} C_VEL
LIN {X 0,Y 433.022,Z 365.168,A -85,B 0,C 180,E1 -9968.207,E2 -9968.207} C_VEL
LIN {X 0,Y 431.857,Z 379.994,A -85,B 0,C 180,E1 -9969.146,E2 -9969.146} C_VEL
LIN {X 0,Y 430.703,Z 393.383,A -85,B 0,C 180,E1 -9970.21,E2 -9970.21} C_VEL
LIN {X 0,Y 429.583,Z 405.652,A -85,B 0,C 180,E1 -9971.397,E2 -9971.397} C_VEL
LIN {X 0,Y 428.351,Z 417.87,A -85,B 0,C 180,E1 -9972.823,E2 -9972.823} C_VEL
LIN {X 0,Y 427.351,Z 428.09,A -85,B 0,C 180,E1 -9974.256,E2 -9974.256} C_VEL
LIN {X 0,Y 426.347,Z 438.094,A -85,B 0,C 180,E1 -9975.929,E2 -9975.929} C_VEL
LIN {X 0,Y 425.643,Z 446.392,A -85,B 0,C 180,E1 -9977.606,E2 -9977.606} C_VEL
LIN {X 0,Y 425.129,Z 452.384,A -85,B 0,C 180,E1 -9979.041,E2 -9979.041} C_VEL
LIN {X 0,Y 424.654,Z 458.976,A -85,B 0,C 180,E1 -9980.955,E2 -9980.955} C_VEL
LIN {X 0,Y 424.336,Z 464.132,A -85,B 0,C 180,E1 -9982.865,E2 -9982.865} C_VEL
LIN {X 0,Y 424.188,Z 467.714,A -85,B 0,C 180,E1 -9984.659,E2 -9984.659} C_VEL
LIN {X 0,Y 424.085,Z 470.014,A -85,B 0,C 180,E1 -9986.2,E2 -9986.2} C_VEL
LIN {X 0,Y 424.126,Z 471.766,A -85,B 0,C 180,E1 -9988.101,E2 -9988.101} C_VEL
LIN {X 0,Y 424.073,Z 472.076,A -85,B 0,C 180,E1 -9988.748,E2 -9988.748} C_VEL
LIN {X 0,Y 423.4,Z 472.365,A -85,B 0,C 180,E1 -9989.54,E2 -9989.54} C_VEL
LIN {X 0,Y 420.574,Z 472.41,A -85,B 0,C 180,E1 -9990.83,E2 -9990.83} C_VEL
LIN {X 0,Y 418.174,Z 472,A -85,B 0,C 180,E1 -9991.869,E2 -9991.869} C_VEL
LIN {X 0,Y 417.119,Z 471.401,A -85,B 0,C 180,E1 -9992.668,E2 -9992.668} C_VEL
LIN {X 0,Y 417.019,Z 471.141,A -85,B 0,C 180,E1 -9992.938,E2 -9992.938} C_VEL
LIN {X 0,Y 417.097,Z 468.919,A -85,B 0,C 180,E1 -9994.833,E2 -9994.833} C_VEL
LIN {X 0,Y 417.231,Z 465.463,A -85,B 0,C 180,E1 -9996.772,E2 -9996.772} C_VEL
LIN {X 0,Y 417.499,Z 460.733,A -85,B 0,C 180,E1 -9998.714,E2 -9998.714} C_VEL
LIN {X 0,Y 417.894,Z 454.606,A -85,B 0,C 180,E1 -10000.661,E2 -10000.661} C_VEL
LIN {X 0,Y 418.574,Z 447.947,A -85,B 0,C 180,E1 -10002.362,E2 -10002.362} C_VEL
LIN {X 0,Y 419.213,Z 439.904,A -85,B 0,C 180,E1 -10004.069,E2 -10004.069} C_VEL
LIN {X 0,Y 420.244,Z 430.255,A -85,B 0,C 180,E1 -10005.769,E2 -10005.769} C_VEL
LIN {X 0,Y 421.268,Z 420.391,A -85,B 0,C 180,E1 -10007.225,E2 -10007.225} C_VEL
LIN {X 0,Y 422.512,Z 408.662,A -85,B 0,C 180,E1 -10008.675,E2 -10008.675} C_VEL
LIN {X 0,Y 423.806,Z 395.701,A -85,B 0,C 180,E1 -10010,E2 -10010} C_VEL
LIN {X 0,Y 424.952,Z 382.83,A -85,B 0,C 180,E1 -10011.082,E2 -10011.082} C_VEL
LIN {X 0,Y 426.216,Z 368.713,A -85,B 0,C 180,E1 -10012.032,E2 -10012.032} C_VEL
LIN {X 0,Y 427.089,Z 354.3,A -85,B 0,C 180,E1 -10012.801,E2 -10012.801} C_VEL
LIN {X 0,Y 426.868,Z 351.882,A -85,B 0,C 180,E1 -10012.933,E2 -10012.933} C_VEL
LIN {X 0,Y 423.373,Z 337.938,A -85,B 0,C 180,E1 -10013.705,E2 -10013.705} C_VEL
LIN {X 0,Y 418.731,Z 322.963,A -85,B 0,C 180,E1 -10014.408,E2 -10014.408} C_VEL
LIN {X 0,Y 417.575,Z 318.92,A -85,B 0,C 180,E1 -10014.6,E2 -10014.6} C_VEL
LIN {X 0,Y 417.768,Z 314.021,A -85,B 0,C 180,E1 -10018.102,E2 -10018.102} C_VEL
LIN {X 0,Y 417.991,Z 309.5,A -85,B 0,C 180,E1 -10021.414,E2 -10021.414} C_VEL
LIN {X 0,Y 418.258,Z 304.992,A -85,B 0,C 180,E1 -10024.841,E2 -10024.841} C_VEL
LIN {X 0,Y 418.456,Z 300.461,A -85,B 0,C 180,E1 -10028.42,E2 -10028.42} C_VEL
LIN {X 0,Y 418.589,Z 297.412,A -85,B 0,C 180,E1 -10030.927,E2 -10030.927} C_VEL
LIN {X 0,Y 418.423,Z 294.139,A -85,B 0,C 180,E1 -10033.76,E2 -10033.76} C_VEL
LIN {X 0,Y 418.245,Z 293.017,A -85,B 0,C 180,E1 -10035.11,E2 -10035.11} C_VEL
LIN {X 0,Y 418.239,Z 293.014,A -85,B 0,C 180,E1 -10037.767,E2 -10037.767} C_VEL
LIN {X 0,Y 418.257,Z 293.012,A -85,B 0,C 180,E1 -10040.618,E2 -10040.618} C_VEL
LIN {X 0,Y 418.241,Z 293.014,A -85,B 0,C 180,E1 -10043.975,E2 -10043.975} C_VEL
LIN {X 0,Y 418.256,Z 293.011,A -85,B 0,C 180,E1 -10047.156,E2 -10047.156} C_VEL
LIN {X 0,Y 418.259,Z 293.013,A -85,B 0,C 180,E1 -10050.837,E2 -10050.837} C_VEL
LIN {X 0,Y 418.235,Z 293.016,A -85,B 0,C 180,E1 -10054.093,E2 -10054.093} C_VEL
LIN {X 0,Y 418.229,Z 293.014,A -85,B 0,C 180,E1 -10057.263,E2 -10057.263} C_VEL
LIN {X 0,Y 418.281,Z 293.007,A -85,B 0,C 180,E1 -10060.364,E2 -10060.364} C_VEL
LIN {X 0,Y 418.314,Z 293.002,A -85,B 0,C 180,E1 -10063.404,E2 -10063.404} C_VEL
LIN {X 0,Y 418.343,Z 292.995,A -85,B 0,C 180,E1 -10066.999,E2 -10066.999} C_VEL
LIN {X 0,Y 418.337,Z 293,A -85,B 0,C 180,E1 -10070.328,E2 -10070.328} C_VEL
LIN {X 0,Y 418.442,Z 292.986,A -85,B 0,C 180,E1 -10073.248,E2 -10073.248} C_VEL
LIN {X 0,Y 418.334,Z 293.002,A -85,B 0,C 180,E1 -10075.181,E2 -10075.181} C_VEL
LIN {X 0,Y 418.542,Z 292.974,A -85,B 0,C 180,E1 -10078.075,E2 -10078.075} C_VEL
LIN {X 0,Y 418.662,Z 292.962,A -85,B 0,C 180,E1 -10080,E2 -10080} C_VEL
LIN {X 0,Y 418.508,Z 292.981,A -85,B 0,C 180,E1 -10082.888,E2 -10082.888} C_VEL
LIN {X 0,Y 418.489,Z 292.981,A -85,B 0,C 180,E1 -10085.783,E2 -10085.783} C_VEL
LIN {X 0,Y 418.375,Z 292.995,A -85,B 0,C 180,E1 -10088.695,E2 -10088.695} C_VEL
LIN {X 0,Y 418.313,Z 293.003,A -85,B 0,C 180,E1 -10091.631,E2 -10091.631} C_VEL
LIN {X 0,Y 418.299,Z 293.005,A -85,B 0,C 180,E1 -10094.597,E2 -10094.597} C_VEL
LIN {X 0,Y 418.285,Z 293.006,A -85,B 0,C 180,E1 -10097.604,E2 -10097.604} C_VEL
LIN {X 0,Y 418.247,Z 293.011,A -85,B 0,C 180,E1 -10100.663,E2 -10100.663} C_VEL
LIN {X 0,Y 418.273,Z 293.007,A -85,B 0,C 180,E1 -10103.782,E2 -10103.782} C_VEL
LIN {X 0,Y 418.308,Z 293.005,A -85,B 0,C 180,E1 -10107.071,E2 -10107.071} C_VEL
LIN {X 0,Y 418.241,Z 293.016,A -85,B 0,C 180,E1 -10110.272,E2 -10110.272} C_VEL
LIN {X 0,Y 418.246,Z 293.019,A -85,B 0,C 180,E1 -10113.677,E2 -10113.677} C_VEL
LIN {X 0,Y 418.237,Z 293.019,A -85,B 0,C 180,E1 -10117.224,E2 -10117.224} C_VEL
LIN {X 0,Y 418.24,Z 293.017,A -85,B 0,C 180,E1 -10119.683,E2 -10119.683} C_VEL
LIN {X 0,Y 418.221,Z 293.017,A -85,B 0,C 180,E1 -10122.32,E2 -10122.32} C_VEL
LIN {X 0,Y 418.366,Z 293.648,A -85,B 0,C 180,E1 -10123.752,E2 -10123.752} C_VEL
LIN {X 0,Y 418.857,Z 297.149,A -85,B 0,C 180,E1 -10126.533,E2 -10126.533} C_VEL
LIN {X 0,Y 419.013,Z 300.645,A -85,B 0,C 180,E1 -10129.146,E2 -10129.146} C_VEL
LIN {X 0,Y 418.814,Z 304.784,A -85,B 0,C 180,E1 -10132.063,E2 -10132.063} C_VEL
LIN {X 0,Y 418.528,Z 309.686,A -85,B 0,C 180,E1 -10135.368,E2 -10135.368} C_VEL
LIN {X 0,Y 418.176,Z 315.303,A -85,B 0,C 180,E1 -10138.995,E2 -10138.995} C_VEL
LIN {X 0,Y 417.874,Z 319.963,A -85,B 0,C 180,E1 -10141.906,E2 -10141.906} C_VEL
LIN {X 0,Y 417.638,Z 325.822,A -85,B 0,C 180,E1 -10145.463,E2 -10145.463} C_VEL
LIN {X 0,Y 422.731,Z 343.425,A -85,B 0,C 180,E1 -10146.229,E2 -10146.229} C_VEL
LIN {X 0,Y 426.082,Z 357.281,A -85,B 0,C 180,E1 -10146.962,E2 -10146.962} C_VEL
LIN {X 0,Y 426.895,Z 361.483,A -85,B 0,C 180,E1 -10147.21,E2 -10147.21} C_VEL
LIN {X 0,Y 426.051,Z 375.692,A -85,B 0,C 180,E1 -10147.959,E2 -10147.959} C_VEL
LIN {X 0,Y 424.853,Z 389.98,A -85,B 0,C 180,E1 -10148.912,E2 -10148.912} C_VEL
LIN {X 0,Y 423.62,Z 402.984,A -85,B 0,C 180,E1 -10149.99,E2 -10149.99} C_VEL
LIN {X 0,Y 422.419,Z 414.99,A -85,B 0,C 180,E1 -10151.195,E2 -10151.195} C_VEL
LIN {X 0,Y 421.318,Z 426.109,A -85,B 0,C 180,E1 -10152.527,E2 -10152.527} C_VEL
LIN {X 0,Y 420.228,Z 436.336,A -85,B 0,C 180,E1 -10153.981,E2 -10153.981} C_VEL
LIN {X 0,Y 419.207,Z 446.331,A -85,B 0,C 180,E1 -10155.683,E2 -10155.683} C_VEL
LIN {X 0,Y 418.439,Z 454.63,A -85,B 0,C 180,E1 -10157.388,E2 -10157.388} C_VEL
LIN {X 0,Y 418.002,Z 460.613,A -85,B 0,C 180,E1 -10158.851,E2 -10158.851} C_VEL
LIN {X 0,Y 417.481,Z 467.199,A -85,B 0,C 180,E1 -10160.797,E2 -10160.797} C_VEL
LIN {X 0,Y 417.238,Z 472.351,A -85,B 0,C 180,E1 -10162.742,E2 -10162.742} C_VEL
LIN {X 0,Y 417.081,Z 475.331,A -85,B 0,C 180,E1 -10164.197,E2 -10164.197} C_VEL
LIN {X 0,Y 416.975,Z 478.234,A -85,B 0,C 180,E1 -10166.134,E2 -10166.134} C_VEL
LIN {X 0,Y 417.026,Z 479.966,A -85,B 0,C 180,E1 -10168.068,E2 -10168.068} C_VEL
LIN {X 0,Y 416.98,Z 480.559,A -85,B 0,C 180,E1 -10170,E2 -10170} C_VEL
LIN {X 0,Y 417.026,Z 479.962,A -85,B 0,C 180,E1 -10171.931,E2 -10171.931} C_VEL
LIN {X 0,Y 416.976,Z 478.226,A -85,B 0,C 180,E1 -10173.865,E2 -10173.865} C_VEL
LIN {X 0,Y 417.1,Z 475.325,A -85,B 0,C 180,E1 -10175.802,E2 -10175.802} C_VEL
LIN {X 0,Y 417.26,Z 471.187,A -85,B 0,C 180,E1 -10177.743,E2 -10177.743} C_VEL
LIN {X 0,Y 417.563,Z 465.703,A -85,B 0,C 180,E1 -10179.689,E2 -10179.689} C_VEL
LIN {X 0,Y 418.189,Z 458.724,A -85,B 0,C 180,E1 -10181.634,E2 -10181.634} C_VEL
LIN {X 0,Y 418.642,Z 452.026,A -85,B 0,C 180,E1 -10183.175,E2 -10183.175} C_VEL
LIN {X 0,Y 419.498,Z 443.601,A -85,B 0,C 180,E1 -10184.802,E2 -10184.802} C_VEL
LIN {X 0,Y 420.516,Z 433.052,A -85,B 0,C 180,E1 -10186.505,E2 -10186.505} C_VEL
LIN {X 0,Y 421.709,Z 422.089,A -85,B 0,C 180,E1 -10187.974,E2 -10187.974} C_VEL
LIN {X 0,Y 422.89,Z 410.397,A -85,B 0,C 180,E1 -10189.286,E2 -10189.286} C_VEL
LIN {X 0,Y 424.103,Z 397.465,A -85,B 0,C 180,E1 -10190.491,E2 -10190.491} C_VEL
LIN {X 0,Y 425.421,Z 383.177,A -85,B 0,C 180,E1 -10191.565,E2 -10191.565} C_VEL
LIN {X 0,Y 426.528,Z 368.856,A -85,B 0,C 180,E1 -10192.418,E2 -10192.418} C_VEL
LIN {X 0,Y 426.887,Z 361.449,A -85,B 0,C 180,E1 -10192.788,E2 -10192.788} C_VEL
LIN {X 0,Y 423.675,Z 347.059,A -85,B 0,C 180,E1 -10193.581,E2 -10193.581} C_VEL
LIN {X 0,Y 419.202,Z 331.399,A -85,B 0,C 180,E1 -10194.305,E2 -10194.305} C_VEL
LIN {X 0,Y 417.641,Z 325.855,A -85,B 0,C 180,E1 -10194.523,E2 -10194.523} C_VEL
LIN {X 0,Y 417.869,Z 320.004,A -85,B 0,C 180,E1 -10198.093,E2 -10198.093} C_VEL
LIN {X 0,Y 418.174,Z 314.748,A -85,B 0,C 180,E1 -10201.398,E2 -10201.398} C_VEL
LIN {X 0,Y 418.54,Z 309.455,A -85,B 0,C 180,E1 -10204.813,E2 -10204.813} C_VEL
LIN {X 0,Y 418.811,Z 304.804,A -85,B 0,C 180,E1 -10207.936,E2 -10207.936} C_VEL
LIN {X 0,Y 419.041,Z 300.436,A -85,B 0,C 180,E1 -10210.999,E2 -10210.999} C_VEL
LIN {X 0,Y 418.804,Z 296.68,A -85,B 0,C 180,E1 -10213.814,E2 -10213.814} C_VEL
LIN {X 0,Y 418.289,Z 293.368,A -85,B 0,C 180,E1 -10216.459,E2 -10216.459} C_VEL
LIN {X 0,Y 418.235,Z 293.016,A -85,B 0,C 180,E1 -10217.766,E2 -10217.766} C_VEL
LIN {X 0,Y 418.247,Z 293.014,A -85,B 0,C 180,E1 -10220.619,E2 -10220.619} C_VEL
LIN {X 0,Y 418.236,Z 293.015,A -85,B 0,C 180,E1 -10223.975,E2 -10223.975} C_VEL
LIN {X 0,Y 418.251,Z 293.015,A -85,B 0,C 180,E1 -10227.156,E2 -10227.156} C_VEL
LIN {X 0,Y 418.261,Z 293.015,A -85,B 0,C 180,E1 -10230.895,E2 -10230.895} C_VEL
LIN {X 0,Y 418.263,Z 293.012,A -85,B 0,C 180,E1 -10234.096,E2 -10234.096} C_VEL
LIN {X 0,Y 418.23,Z 293.015,A -85,B 0,C 180,E1 -10237.264,E2 -10237.264} C_VEL
LIN {X 0,Y 418.275,Z 293.009,A -85,B 0,C 180,E1 -10240.364,E2 -10240.364} C_VEL
LIN {X 0,Y 418.309,Z 293.005,A -85,B 0,C 180,E1 -10243.404,E2 -10243.404} C_VEL
LIN {X 0,Y 418.338,Z 292.999,A -85,B 0,C 180,E1 -10246.999,E2 -10246.999} C_VEL
LIN {X 0,Y 418.333,Z 293,A -85,B 0,C 180,E1 -10250.329,E2 -10250.329} C_VEL
LIN {X 0,Y 418.437,Z 292.987,A -85,B 0,C 180,E1 -10253.248,E2 -10253.248} C_VEL
LIN {X 0,Y 418.332,Z 293,A -85,B 0,C 180,E1 -10255.182,E2 -10255.182} C_VEL
LIN {X 0,Y 418.537,Z 292.972,A -85,B 0,C 180,E1 -10258.076,E2 -10258.076} C_VEL
LIN {X 0,Y 418.659,Z 292.963,A -85,B 0,C 180,E1 -10260,E2 -10260} C_VEL
LIN {X 0,Y 418.504,Z 292.981,A -85,B 0,C 180,E1 -10262.888,E2 -10262.888} C_VEL
LIN {X 0,Y 418.439,Z 292.986,A -85,B 0,C 180,E1 -10266.454,E2 -10266.454} C_VEL
LIN {X 0,Y 418.332,Z 293.001,A -85,B 0,C 180,E1 -10269.672,E2 -10269.672} C_VEL
LIN {X 0,Y 418.338,Z 292.999,A -85,B 0,C 180,E1 -10273.001,E2 -10273.001} C_VEL
LIN {X 0,Y 418.305,Z 293.007,A -85,B 0,C 180,E1 -10276.736,E2 -10276.736} C_VEL
LIN {X 0,Y 418.263,Z 293.012,A -85,B 0,C 180,E1 -10279.791,E2 -10279.791} C_VEL
LIN {X 0,Y 418.231,Z 293.015,A -85,B 0,C 180,E1 -10282.737,E2 -10282.737} C_VEL
LIN {X 0,Y 418.264,Z 293.011,A -85,B 0,C 180,E1 -10285.905,E2 -10285.905} C_VEL
LIN {X 0,Y 418.258,Z 293.01,A -85,B 0,C 180,E1 -10289.163,E2 -10289.163} C_VEL
LIN {X 0,Y 418.251,Z 293.007,A -85,B 0,C 180,E1 -10292.845,E2 -10292.845} C_VEL
LIN {X 0,Y 418.239,Z 293.011,A -85,B 0,C 180,E1 -10296.239,E2 -10296.239} C_VEL
LIN {X 0,Y 418.249,Z 293.014,A -85,B 0,C 180,E1 -10299.682,E2 -10299.682} C_VEL
LIN {X 0,Y 418.225,Z 293.016,A -85,B 0,C 180,E1 -10302.322,E2 -10302.322} C_VEL
LIN {X 0,Y 418.232,Z 293.014,A -85,B 0,C 180,E1 -10305.11,E2 -10305.11} C_VEL
LIN {X 0,Y 418.51,Z 295.596,A -85,B 0,C 180,E1 -10307.637,E2 -10307.637} C_VEL
LIN {X 0,Y 418.553,Z 298.796,A -85,B 0,C 180,E1 -10310.354,E2 -10310.354} C_VEL
LIN {X 0,Y 418.313,Z 303.304,A -85,B 0,C 180,E1 -10313.984,E2 -10313.984} C_VEL
LIN {X 0,Y 418.077,Z 307.444,A -85,B 0,C 180,E1 -10317.195,E2 -10317.195} C_VEL
LIN {X 0,Y 417.913,Z 310.81,A -85,B 0,C 180,E1 -10319.702,E2 -10319.702} C_VEL
LIN {X 0,Y 417.692,Z 315.499,A -85,B 0,C 180,E1 -10323.096,E2 -10323.096} C_VEL
LIN {X 0,Y 417.597,Z 319.106,A -85,B 0,C 180,E1 -10325.536,E2 -10325.536} C_VEL
LIN {X 0,Y 422.647,Z 335.358,A -85,B 0,C 180,E1 -10326.256,E2 -10326.256} C_VEL
LIN {X 0,Y 426.347,Z 349.681,A -85,B 0,C 180,E1 -10327.028,E2 -10327.028} C_VEL
LIN {X 0,Y 427.148,Z 353.975,A -85,B 0,C 180,E1 -10327.281,E2 -10327.281} C_VEL
LIN {X 0,Y 426.125,Z 369.22,A -85,B 0,C 180,E1 -10328.091,E2 -10328.091} C_VEL
LIN {X 0,Y 424.9,Z 383.23,A -85,B 0,C 180,E1 -10329.043,E2 -10329.043} C_VEL
LIN {X 0,Y 423.745,Z 396.037,A -85,B 0,C 180,E1 -10330.124,E2 -10330.124} C_VEL
LIN {X 0,Y 422.573,Z 408.087,A -85,B 0,C 180,E1 -10331.354,E2 -10331.354} C_VEL
LIN {X 0,Y 421.323,Z 419.725,A -85,B 0,C 180,E1 -10332.778,E2 -10332.778} C_VEL
LIN {X 0,Y 420.313,Z 429.698,A -85,B 0,C 180,E1 -10334.234,E2 -10334.234} C_VEL
LIN {X 0,Y 419.3,Z 439.439,A -85,B 0,C 180,E1 -10335.935,E2 -10335.935} C_VEL
LIN {X 0,Y 418.596,Z 447.558,A -85,B 0,C 180,E1 -10337.64,E2 -10337.64} C_VEL
LIN {X 0,Y 417.918,Z 454.26,A -85,B 0,C 180,E1 -10339.34,E2 -10339.34} C_VEL
LIN {X 0,Y 417.514,Z 460.467,A -85,B 0,C 180,E1 -10341.287,E2 -10341.287} C_VEL
LIN {X 0,Y 417.23,Z 465.262,A -85,B 0,C 180,E1 -10343.229,E2 -10343.229} C_VEL
LIN {X 0,Y 417.101,Z 468.776,A -85,B 0,C 180,E1 -10345.168,E2 -10345.168} C_VEL
LIN {X 0,Y 417.022,Z 471.101,A -85,B 0,C 180,E1 -10347.102,E2 -10347.102} C_VEL
LIN {X 0,Y 416.991,Z 472.29,A -85,B 0,C 180,E1 -10349.035,E2 -10349.035} C_VEL
LIN {X 0,Y 416.991,Z 472.306,A -85,B 0,C 180,E1 -10350.966,E2 -10350.966} C_VEL
LIN {X 0,Y 417.019,Z 471.141,A -85,B 0,C 180,E1 -10352.938,E2 -10352.938} C_VEL
LIN {X 0,Y 416.329,Z 470.37,A -85,B 0,C 180,E1 -10353.736,E2 -10353.736} C_VEL
LIN {X 0,Y 413.533,Z 468.724,A -85,B 0,C 180,E1 -10355.03,E2 -10355.03} C_VEL
LIN {X 0,Y 411.209,Z 467.091,A -85,B 0,C 180,E1 -10356.065,E2 -10356.065} C_VEL
LIN {X 0,Y 410.237,Z 465.607,A -85,B 0,C 180,E1 -10356.855,E2 -10356.855} C_VEL
LIN {X 0,Y 410.169,Z 465.034,A -85,B 0,C 180,E1 -10357.121,E2 -10357.121} C_VEL
LIN {X 0,Y 410.443,Z 460.801,A -85,B 0,C 180,E1 -10358.865,E2 -10358.865} C_VEL
LIN {X 0,Y 410.878,Z 454.673,A -85,B 0,C 180,E1 -10360.845,E2 -10360.845} C_VEL
LIN {X 0,Y 411.556,Z 448.014,A -85,B 0,C 180,E1 -10362.576,E2 -10362.576} C_VEL
LIN {X 0,Y 412.435,Z 438.735,A -85,B 0,C 180,E1 -10364.557,E2 -10364.557} C_VEL
LIN {X 0,Y 413.519,Z 428.832,A -85,B 0,C 180,E1 -10366.286,E2 -10366.286} C_VEL
LIN {X 0,Y 414.718,Z 418.678,A -85,B 0,C 180,E1 -10367.76,E2 -10367.76} C_VEL
LIN {X 0,Y 416.015,Z 406.592,A -85,B 0,C 180,E1 -10369.234,E2 -10369.234} C_VEL
LIN {X 0,Y 417.136,Z 395.765,A -85,B 0,C 180,E1 -10370.334,E2 -10370.334} C_VEL
LIN {X 0,Y 418.3,Z 382.894,A -85,B 0,C 180,E1 -10371.434,E2 -10371.434} C_VEL
LIN {X 0,Y 419.615,Z 368.775,A -85,B 0,C 180,E1 -10372.398,E2 -10372.398} C_VEL
LIN {X 0,Y 420.487,Z 354.344,A -85,B 0,C 180,E1 -10373.18,E2 -10373.18} C_VEL
LIN {X 0,Y 416.943,Z 339.965,A -85,B 0,C 180,E1 -10374.022,E2 -10374.022} C_VEL
LIN {X 0,Y 412.452,Z 325.091,A -85,B 0,C 180,E1 -10374.758,E2 -10374.758} C_VEL
LIN {X 0,Y 410.512,Z 319.024,A -85,B 0,C 180,E1 -10375.027,E2 -10375.027} C_VEL
LIN {X 0,Y 410.731,Z 314.08,A -85,B 0,C 180,E1 -10378.627,E2 -10378.627} C_VEL
LIN {X 0,Y 411.004,Z 309.573,A -85,B 0,C 180,E1 -10382.011,E2 -10382.011} C_VEL
LIN {X 0,Y 411.255,Z 305.053,A -85,B 0,C 180,E1 -10385.523,E2 -10385.523} C_VEL
LIN {X 0,Y 411.492,Z 300.519,A -85,B 0,C 180,E1 -10389.193,E2 -10389.193} C_VEL
LIN {X 0,Y 411.538,Z 297.492,A -85,B 0,C 180,E1 -10391.76,E2 -10391.76} C_VEL
LIN {X 0,Y 411.279,Z 294.453,A -85,B 0,C 180,E1 -10394.476,E2 -10394.476} C_VEL
LIN {X 0,Y 411.17,Z 293.898,A -85,B 0,C 180,E1 -10395.88,E2 -10395.88} C_VEL
LIN {X 0,Y 411.164,Z 293.897,A -85,B 0,C 180,E1 -10398.771,E2 -10398.771} C_VEL
LIN {X 0,Y 411.206,Z 293.893,A -85,B 0,C 180,E1 -10401.831,E2 -10401.831} C_VEL
LIN {X 0,Y 411.209,Z 293.892,A -85,B 0,C 180,E1 -10405.121,E2 -10405.121} C_VEL
LIN {X 0,Y 411.163,Z 293.897,A -85,B 0,C 180,E1 -10408.002,E2 -10408.002} C_VEL
LIN {X 0,Y 411.192,Z 293.891,A -85,B 0,C 180,E1 -10411.408,E2 -10411.408} C_VEL
LIN {X 0,Y 411.224,Z 293.886,A -85,B 0,C 180,E1 -10414.929,E2 -10414.929} C_VEL
LIN {X 0,Y 411.202,Z 293.886,A -85,B 0,C 180,E1 -10417.913,E2 -10417.913} C_VEL
